LIN {X 0,Y 417.016,Z 398.719,A -85,B 0,C 180,E1 -10166.134,E2 -10166.134} C_VEL
LIN {X 0,Y 417.047,Z 400.246,A -85,B 0,C 180,E1 -10167.102,E2 -10167.102} C_VEL
LIN {X 0,Y 417.071,Z 401.315,A -85,B 0,C 180,E1 -10168.068,E2 -10168.068} C_VEL
LIN {X 0,Y 417.03,Z 402.263,A -85,B 0,C 180,E1 -10170,E2 -10170} C_VEL
LIN {X 0,Y 417.016,Z 402.15,A -85,B 0,C 180,E1 -10170.965,E2 -10170.965} C_VEL
LIN {X 0,Y 417.07,Z 401.605,A -85,B 0,C 180,E1 -10171.931,E2 -10171.931} C_VEL
LIN {X 0,Y 417.03,Z 400.658,A -85,B 0,C 180,E1 -10172.898,E2 -10172.898} C_VEL
LIN {X 0,Y 417.014,Z 399.317,A -85,B 0,C 180,E1 -10173.865,E2 -10173.865} C_VEL
LIN {X 0,Y 417.113,Z 396.49,A -85,B 0,C 180,E1 -10175.317,E2 -10175.317} C_VEL
LIN {X 0,Y 417.163,Z 392.636,A -85,B 0,C 180,E1 -10176.773,E2 -10176.773} C_VEL
LIN {X 0,Y 417.446,Z 387.665,A -85,B 0,C 180,E1 -10178.227,E2 -10178.227} C_VEL
LIN {X 0,Y 417.809,Z 381.424,A -85,B 0,C 180,E1 -10179.684,E2 -10179.684} C_VEL
LIN {X 0,Y 418.374,Z 373.662,A -85,B 0,C 180,E1 -10181.138,E2 -10181.138} C_VEL
LIN {X 0,Y 419.211,Z 363.972,A -85,B 0,C 180,E1 -10182.588,E2 -10182.588} C_VEL
LIN {X 0,Y 419.889,Z 353.988,A -85,B 0,C 180,E1 -10183.799,E2 -10183.799} C_VEL
LIN {X 0,Y 420.769,Z 342.734,A -85,B 0,C 180,E1 -10184.881,E2 -10184.881} C_VEL
LIN {X 0,Y 421.539,Z 331.733,A -85,B 0,C 180,E1 -10185.719,E2 -10185.719} C_VEL
LIN {X 0,Y 422.358,Z 319.563,A -85,B 0,C 180,E1 -10186.432,E2 -10186.432} C_VEL
LIN {X 0,Y 422.975,Z 306.851,A -85,B 0,C 180,E1 -10186.966,E2 -10186.966} C_VEL
LIN {X 0,Y 423.495,Z 293.508,A -85,B 0,C 180,E1 -10187.318,E2 -10187.318} C_VEL
LIN {X 0,Y 424.284,Z 215.513,A -85,B 0,C 180,E1 -10188.688,E2 -10188.688} C_VEL
LIN {X 0,Y 421.243,Z 196.282,A -85,B 0,C 180,E1 -10189.197,E2 -10189.197} C_VEL
LIN {X 0,Y 419.891,Z 188.95,A -85,B 0,C 180,E1 -10189.422,E2 -10189.422} C_VEL
LIN {X 0,Y 421.037,Z 171.63,A -85,B 0,C 180,E1 -10192.794,E2 -10192.794} C_VEL
LIN {X 0,Y 421.61,Z 163.663,A -85,B 0,C 180,E1 -10194.366,E2 -10194.366} C_VEL
LIN {X 0,Y 420.366,Z 155.936,A -85,B 0,C 180,E1 -10196.032,E2 -10196.032} C_VEL
LIN {X 0,Y 418.252,Z 146.389,A -85,B 0,C 180,E1 -10198.203,E2 -10198.203} C_VEL
LIN {X 0,Y 418.213,Z 146.395,A -85,B 0,C 180,E1 -10201.396,E2 -10201.396} C_VEL
LIN {X 0,Y 418.255,Z 146.379,A -85,B 0,C 180,E1 -10204.577,E2 -10204.577} C_VEL
LIN {X 0,Y 418.222,Z 146.388,A -85,B 0,C 180,E1 -10207.832,E2 -10207.832} C_VEL
LIN {X 0,Y 418.209,Z 146.385,A -85,B 0,C 180,E1 -10210.95,E2 -10210.95} C_VEL
LIN {X 0,Y 418.205,Z 146.389,A -85,B 0,C 180,E1 -10213.728,E2 -10213.728} C_VEL
LIN {X 0,Y 418.201,Z 146.391,A -85,B 0,C 180,E1 -10216.447,E2 -10216.447} C_VEL
LIN {X 0,Y 418.208,Z 146.39,A -85,B 0,C 180,E1 -10219.133,E2 -10219.133} C_VEL
LIN {X 0,Y 418.233,Z 146.387,A -85,B 0,C 180,E1 -10222.775,E2 -10222.775} C_VEL
LIN {X 0,Y 418.229,Z 146.384,A -85,B 0,C 180,E1 -10226.321,E2 -10226.321} C_VEL
LIN {X 0,Y 418.235,Z 146.38,A -85,B 0,C 180,E1 -10229.727,E2 -10229.727} C_VEL
LIN {X 0,Y 418.203,Z 146.384,A -85,B 0,C 180,E1 -10233.016,E2 -10233.016} C_VEL
LIN {X 0,Y 418.253,Z 146.386,A -85,B 0,C 180,E1 -10236.216,E2 -10236.216} C_VEL
LIN {X 0,Y 418.23,Z 146.385,A -85,B 0,C 180,E1 -10239.335,E2 -10239.335} C_VEL
LIN {X 0,Y 418.237,Z 146.383,A -85,B 0,C 180,E1 -10242.394,E2 -10242.394} C_VEL
LIN {X 0,Y 418.279,Z 146.38,A -85,B 0,C 180,E1 -10245.402,E2 -10245.402} C_VEL
LIN {X 0,Y 418.307,Z 146.379,A -85,B 0,C 180,E1 -10248.368,E2 -10248.368} C_VEL
LIN {X 0,Y 418.449,Z 146.356,A -85,B 0,C 180,E1 -10252.278,E2 -10252.278} C_VEL
LIN {X 0,Y 418.487,Z 146.355,A -85,B 0,C 180,E1 -10254.216,E2 -10254.216} C_VEL
LIN {X 0,Y 418.536,Z 146.349,A -85,B 0,C 180,E1 -10258.075,E2 -10258.075} C_VEL
LIN {X 0,Y 418.565,Z 146.342,A -85,B 0,C 180,E1 -10259.999,E2 -10259.999} C_VEL
LIN {X 0,Y 418.493,Z 146.351,A -85,B 0,C 180,E1 -10262.887,E2 -10262.887} C_VEL
LIN {X 0,Y 418.446,Z 146.353,A -85,B 0,C 180,E1 -10266.519,E2 -10266.519} C_VEL
LIN {X 0,Y 418.34,Z 146.369,A -85,B 0,C 180,E1 -10269.671,E2 -10269.671} C_VEL
LIN {X 0,Y 418.348,Z 146.376,A -85,B 0,C 180,E1 -10273,E2 -10273} C_VEL
LIN {X 0,Y 418.313,Z 146.378,A -85,B 0,C 180,E1 -10276.734,E2 -10276.734} C_VEL
LIN {X 0,Y 418.271,Z 146.382,A -85,B 0,C 180,E1 -10279.789,E2 -10279.789} C_VEL
LIN {X 0,Y 418.232,Z 146.387,A -85,B 0,C 180,E1 -10282.736,E2 -10282.736} C_VEL
LIN {X 0,Y 418.261,Z 146.383,A -85,B 0,C 180,E1 -10285.904,E2 -10285.904} C_VEL
LIN {X 0,Y 418.268,Z 146.385,A -85,B 0,C 180,E1 -10289.104,E2 -10289.104} C_VEL
LIN {X 0,Y 418.256,Z 146.386,A -85,B 0,C 180,E1 -10292.843,E2 -10292.843} C_VEL
LIN {X 0,Y 418.243,Z 146.391,A -85,B 0,C 180,E1 -10296.237,E2 -10296.237} C_VEL
LIN {X 0,Y 418.247,Z 146.387,A -85,B 0,C 180,E1 -10299.682,E2 -10299.682} C_VEL
LIN {X 0,Y 418.228,Z 146.392,A -85,B 0,C 180,E1 -10302.321,E2 -10302.321} C_VEL
LIN {X 0,Y 418.234,Z 146.39,A -85,B 0,C 180,E1 -10305.108,E2 -10305.108} C_VEL
LIN {X 0,Y 418.247,Z 146.493,A -85,B 0,C 180,E1 -10307.098,E2 -10307.098} C_VEL
LIN {X 0,Y 420.308,Z 156.513,A -85,B 0,C 180,E1 -10309.56,E2 -10309.56} C_VEL
LIN {X 0,Y 420.473,Z 161.32,A -85,B 0,C 180,E1 -10310.665,E2 -10310.665} C_VEL
LIN {X 0,Y 424.772,Z 180.68,A -85,B 0,C 180,E1 -10311.261,E2 -10311.261} C_VEL
LIN {X 0,Y 423.613,Z 268.691,A -85,B 0,C 180,E1 -10312.816,E2 -10312.816} C_VEL
LIN {X 0,Y 423.211,Z 281.385,A -85,B 0,C 180,E1 -10313.221,E2 -10313.221} C_VEL
LIN {X 0,Y 422.69,Z 294.104,A -85,B 0,C 180,E1 -10313.825,E2 -10313.825} C_VEL
LIN {X 0,Y 421.974,Z 306.065,A -85,B 0,C 180,E1 -10314.596,E2 -10314.596} C_VEL
LIN {X 0,Y 421.162,Z 317.748,A -85,B 0,C 180,E1 -10315.578,E2 -10315.578} C_VEL
LIN {X 0,Y 420.343,Z 328.498,A -85,B 0,C 180,E1 -10316.717,E2 -10316.717} C_VEL
LIN {X 0,Y 419.641,Z 337.311,A -85,B 0,C 180,E1 -10317.877,E2 -10317.877} C_VEL
LIN {X 0,Y 418.911,Z 345.664,A -85,B 0,C 180,E1 -10319.223,E2 -10319.223} C_VEL
LIN {X 0,Y 418.274,Z 353.696,A -85,B 0,C 180,E1 -10320.839,E2 -10320.839} C_VEL
LIN {X 0,Y 417.818,Z 359.91,A -85,B 0,C 180,E1 -10322.447,E2 -10322.447} C_VEL
LIN {X 0,Y 417.449,Z 364.645,A -85,B 0,C 180,E1 -10324.041,E2 -10324.041} C_VEL
LIN {X 0,Y 417.257,Z 367.76,A -85,B 0,C 180,E1 -10325.44,E2 -10325.44} C_VEL
LIN {X 0,Y 417.028,Z 370.384,A -85,B 0,C 180,E1 -10327.194,E2 -10327.194} C_VEL
LIN {X 0,Y 417.008,Z 371.33,A -85,B 0,C 180,E1 -10328.237,E2 -10328.237} C_VEL
LIN {X 0,Y 416.93,Z 371.775,A -85,B 0,C 180,E1 -10329.269,E2 -10329.269} C_VEL
LIN {X 0,Y 416.941,Z 371.672,A -85,B 0,C 180,E1 -10330.722,E2 -10330.722} C_VEL
LIN {X 0,Y 416.976,Z 370.485,A -85,B 0,C 180,E1 -10332.339,E2 -10332.339} C_VEL
LIN {X 0,Y 417.129,Z 368.427,A -85,B 0,C 180,E1 -10333.812,E2 -10333.812} C_VEL
LIN {X 0,Y 417.298,Z 365.169,A -85,B 0,C 180,E1 -10335.367,E2 -10335.367} C_VEL
LIN {X 0,Y 417.539,Z 360.89,A -85,B 0,C 180,E1 -10336.866,E2 -10336.866} C_VEL
LIN {X 0,Y 417.912,Z 354.367,A -85,B 0,C 180,E1 -10338.603,E2 -10338.603} C_VEL
LIN {X 0,Y 418.368,Z 347.237,A -85,B 0,C 180,E1 -10340.085,E2 -10340.085} C_VEL
LIN {X 0,Y 418.677,Z 342.718,A -85,B 0,C 180,E1 -10340.871,E2 -10340.871} C_VEL
LIN {X 0,Y 418.226,Z 338.947,A -85,B 0,C 180,E1 -10341.486,E2 -10341.486} C_VEL
LIN {X 0,Y 415.824,Z 332.509,A -85,B 0,C 180,E1 -10342.469,E2 -10342.469} C_VEL
LIN {X 0,Y 413.531,Z 325.54,A -85,B 0,C 180,E1 -10343.39,E2 -10343.39} C_VEL
LIN {X 0,Y 413.248,Z 320.905,A -85,B 0,C 180,E1 -10343.904,E2 -10343.904} C_VEL
LIN {X 0,Y 413.946,Z 310.162,A -85,B 0,C 180,E1 -10344.886,E2 -10344.886} C_VEL
LIN {X 0,Y 414.53,Z 298.105,A -85,B 0,C 180,E1 -10345.746,E2 -10345.746} C_VEL
LIN {X 0,Y 415.093,Z 284.913,A -85,B 0,C 180,E1 -10346.448,E2 -10346.448} C_VEL
LIN {X 0,Y 415.474,Z 272.537,A -85,B 0,C 180,E1 -10346.899,E2 -10346.899} C_VEL
LIN {X 0,Y 415.743,Z 256.003,A -85,B 0,C 180,E1 -10347.248,E2 -10347.248} C_VEL
LIN {X 0,Y 416.545,Z 180.606,A -85,B 0,C 180,E1 -10348.565,E2 -10348.565} C_VEL
LIN {X 0,Y 412.854,Z 161.197,A -85,B 0,C 180,E1 -10349.086,E2 -10349.086} C_VEL
LIN {X 0,Y 412.939,Z 156.063,A -85,B 0,C 180,E1 -10350.244,E2 -10350.244} C_VEL
LIN {X 0,Y 411.456,Z 147.236,A -85,B 0,C 180,E1 -10352.386,E2 -10352.386} C_VEL
LIN {X 0,Y 411.411,Z 147.241,A -85,B 0,C 180,E1 -10355.883,E2 -10355.883} C_VEL
LIN {X 0,Y 411.302,Z 147.247,A -85,B 0,C 180,E1 -10358.847,E2 -10358.847} C_VEL
LIN {X 0,Y 411.266,Z 147.259,A -85,B 0,C 180,E1 -10361.834,E2 -10361.834} C_VEL
LIN {X 0,Y 411.203,Z 147.26,A -85,B 0,C 180,E1 -10364.855,E2 -10364.855} C_VEL
LIN {X 0,Y 411.17,Z 147.268,A -85,B 0,C 180,E1 -10367.919,E2 -10367.919} C_VEL
LIN {X 0,Y 411.175,Z 147.265,A -85,B 0,C 180,E1 -10371.036,E2 -10371.036} C_VEL
LIN {X 0,Y 411.167,Z 147.265,A -85,B 0,C 180,E1 -10374.219,E2 -10374.219} C_VEL
LIN {X 0,Y 411.137,Z 147.274,A -85,B 0,C 180,E1 -10377.487,E2 -10377.487} C_VEL
LIN {X 0,Y 411.189,Z 147.264,A -85,B 0,C 180,E1 -10379.714,E2 -10379.714} C_VEL
LIN {X 0,Y 411.2,Z 147.266,A -85,B 0,C 180,E1 -10383.157,E2 -10383.157} C_VEL
LIN {X 0,Y 411.185,Z 147.263,A -85,B 0,C 180,E1 -10386.552,E2 -10386.552} C_VEL
LIN {X 0,Y 411.165,Z 147.266,A -85,B 0,C 180,E1 -10389.721,E2 -10389.721} C_VEL
LIN {X 0,Y 411.159,Z 147.271,A -85,B 0,C 180,E1 -10393.136,E2 -10393.136} C_VEL
LIN {X 0,Y 411.162,Z 147.265,A -85,B 0,C 180,E1 -10395.883,E2 -10395.883} C_VEL
LIN {X 0,Y 411.157,Z 147.266,A -85,B 0,C 180,E1 -10399.494,E2 -10399.494} C_VEL
LIN {X 0,Y 411.181,Z 147.263,A -85,B 0,C 180,E1 -10402.026,E2 -10402.026} C_VEL
LIN {X 0,Y 411.2,Z 147.263,A -85,B 0,C 180,E1 -10405.125,E2 -10405.125} C_VEL
LIN {X 0,Y 411.154,Z 147.267,A -85,B 0,C 180,E1 -10408.002,E2 -10408.002} C_VEL
LIN {X 0,Y 411.168,Z 147.264,A -85,B 0,C 180,E1 -10411.407,E2 -10411.407} C_VEL
LIN {X 0,Y 411.188,Z 147.264,A -85,B 0,C 180,E1 -10414.942,E2 -10414.942} C_VEL
LIN {X 0,Y 411.198,Z 147.263,A -85,B 0,C 180,E1 -10417.914,E2 -10417.914} C_VEL
LIN {X 0,Y 411.18,Z 147.263,A -85,B 0,C 180,E1 -10421.05,E2 -10421.05} C_VEL
LIN {X 0,Y 411.199,Z 147.266,A -85,B 0,C 180,E1 -10424.13,E2 -10424.13} C_VEL
LIN {X 0,Y 411.299,Z 147.248,A -85,B 0,C 180,E1 -10427.166,E2 -10427.166} C_VEL
LIN {X 0,Y 411.278,Z 147.257,A -85,B 0,C 180,E1 -10430.161,E2 -10430.161} C_VEL
LIN {X 0,Y 411.394,Z 147.236,A -85,B 0,C 180,E1 -10433.132,E2 -10433.132} C_VEL
LIN {X 0,Y 411.288,Z 147.249,A -85,B 0,C 180,E1 -10435.099,E2 -10435.099} C_VEL
LIN {X 0,Y 411.506,Z 147.227,A -85,B 0,C 180,E1 -10438.043,E2 -10438.043} C_VEL
LIN {X 0,Y 411.381,Z 147.238,A -85,B 0,C 180,E1 -10440.979,E2 -10440.979} C_VEL
LIN {X 0,Y 411.43,Z 147.232,A -85,B 0,C 180,E1 -10442.938,E2 -10442.938} C_VEL
LIN {X 0,Y 411.393,Z 147.236,A -85,B 0,C 180,E1 -10446.869,E2 -10446.869} C_VEL
LIN {X 0,Y 411.287,Z 147.254,A -85,B 0,C 180,E1 -10449.839,E2 -10449.839} C_VEL
LIN {X 0,Y 411.311,Z 147.249,A -85,B 0,C 180,E1 -10453.104,E2 -10453.104} C_VEL
LIN {X 0,Y 411.215,Z 147.26,A -85,B 0,C 180,E1 -10456.891,E2 -10456.891} C_VEL
LIN {X 0,Y 411.215,Z 147.259,A -85,B 0,C 180,E1 -10459.988,E2 -10459.988} C_VEL
LIN {X 0,Y 411.192,Z 147.267,A -85,B 0,C 180,E1 -10463.149,E2 -10463.149} C_VEL
LIN {X 0,Y 411.176,Z 147.263,A -85,B 0,C 180,E1 -10466.386,E2 -10466.386} C_VEL
LIN {X 0,Y 411.199,Z 147.261,A -85,B 0,C 180,E1 -10469.713,E2 -10469.713} C_VEL
LIN {X 0,Y 411.209,Z 147.264,A -85,B 0,C 180,E1 -10473.156,E2 -10473.156} C_VEL
LIN {X 0,Y 411.196,Z 147.264,A -85,B 0,C 180,E1 -10476.552,E2 -10476.552} C_VEL
LIN {X 0,Y 411.182,Z 147.263,A -85,B 0,C 180,E1 -10479.722,E2 -10479.722} C_VEL
LIN {X 0,Y 411.166,Z 147.267,A -85,B 0,C 180,E1 -10483.135,E2 -10483.135} C_VEL
LIN {X 0,Y 411.168,Z 147.264,A -85,B 0,C 180,E1 -10485.882,E2 -10485.882} C_VEL
LIN {X 0,Y 411.162,Z 147.265,A -85,B 0,C 180,E1 -10489.493,E2 -10489.493} C_VEL
LIN {X 0,Y 411.19,Z 147.263,A -85,B 0,C 180,E1 -10492.025,E2 -10492.025} C_VEL
LIN {X 0,Y 411.207,Z 147.26,A -85,B 0,C 180,E1 -10495.123,E2 -10495.123} C_VEL
LIN {X 0,Y 411.168,Z 147.267,A -85,B 0,C 180,E1 -10498.002,E2 -10498.002} C_VEL
LIN {X 0,Y 411.2,Z 147.264,A -85,B 0,C 180,E1 -10501.408,E2 -10501.408} C_VEL
LIN {X 0,Y 411.229,Z 147.314,A -85,B 0,C 180,E1 -10502.451,E2 -10502.451} C_VEL
LIN {X 0,Y 413.944,Z 161.206,A -85,B 0,C 180,E1 -10505.42,E2 -10505.42} C_VEL
LIN {X 0,Y 413.846,Z 166.622,A -85,B 0,C 180,E1 -10506.498,E2 -10506.498} C_VEL
LIN {X 0,Y 412.705,Z 184.992,A -85,B 0,C 180,E1 -10510.087,E2 -10510.087} C_VEL
LIN {X 0,Y 412.413,Z 189.335,A -85,B 0,C 180,E1 -10510.929,E2 -10510.929} C_VEL
LIN {X 0,Y 416.326,Z 217.289,A -85,B 0,C 180,E1 -10511.589,E2 -10511.589} C_VEL
LIN {X 0,Y 415.353,Z 298.398,A -85,B 0,C 180,E1 -10513.029,E2 -10513.029} C_VEL
LIN {X 0,Y 414.814,Z 312.207,A -85,B 0,C 180,E1 -10513.482,E2 -10513.482} C_VEL
LIN {X 0,Y 414.202,Z 325.137,A -85,B 0,C 180,E1 -10514.121,E2 -10514.121} C_VEL
LIN {X 0,Y 413.45,Z 337.732,A -85,B 0,C 180,E1 -10514.976,E2 -10514.976} C_VEL
LIN {X 0,Y 412.691,Z 349.444,A -85,B 0,C 180,E1 -10516.003,E2 -10516.003} C_VEL
LIN {X 0,Y 411.952,Z 360.048,A -85,B 0,C 180,E1 -10517.186,E2 -10517.186} C_VEL
LIN {X 0,Y 411.37,Z 369.023,A -85,B 0,C 180,E1 -10518.419,E2 -10518.419} C_VEL
LIN {X 0,Y 410.782,Z 377.769,A -85,B 0,C 180,E1 -10519.9,E2 -10519.9} C_VEL
LIN {X 0,Y 410.39,Z 384.734,A -85,B 0,C 180,E1 -10521.382,E2 -10521.382} C_VEL
LIN {X 0,Y 410.095,Z 391.121,A -85,B 0,C 180,E1 -10523.11,E2 -10523.11} C_VEL
LIN {X 0,Y 410.004,Z 395.299,A -85,B 0,C 180,E1 -10524.59,E2 -10524.59} C_VEL
LIN {X 0,Y 409.935,Z 398.402,A -85,B 0,C 180,E1 -10526.068,E2 -10526.068} C_VEL
LIN {X 0,Y 409.946,Z 399.944,A -85,B 0,C 180,E1 -10527.052,E2 -10527.052} C_VEL
LIN {X 0,Y 409.999,Z 401.03,A -85,B 0,C 180,E1 -10528.035,E2 -10528.035} C_VEL
LIN {X 0,Y 409.951,Z 401.998,A -85,B 0,C 180,E1 -10530,E2 -10530} C_VEL
LIN {X 0,Y 409.941,Z 401.899,A -85,B 0,C 180,E1 -10530.982,E2 -10530.982} C_VEL
LIN {X 0,Y 409.997,Z 401.37,A -85,B 0,C 180,E1 -10531.965,E2 -10531.965} C_VEL
LIN {X 0,Y 409.932,Z 399.1,A -85,B 0,C 180,E1 -10533.932,E2 -10533.932} C_VEL
LIN {X 0,Y 410.006,Z 396.296,A -85,B 0,C 180,E1 -10535.41,E2 -10535.41} C_VEL
LIN {X 0,Y 410.084,Z 392.472,A -85,B 0,C 180,E1 -10536.89,E2 -10536.89} C_VEL
LIN {X 0,Y 410.402,Z 387.537,A -85,B 0,C 180,E1 -10538.37,E2 -10538.37} C_VEL
LIN {X 0,Y 410.786,Z 381.34,A -85,B 0,C 180,E1 -10539.851,E2 -10539.851} C_VEL
LIN {X 0,Y 411.396,Z 373.648,A -85,B 0,C 180,E1 -10541.33,E2 -10541.33} C_VEL
LIN {X 0,Y 412.279,Z 364.011,A -85,B 0,C 180,E1 -10542.803,E2 -10542.803} C_VEL
LIN {X 0,Y 413.037,Z 353.536,A -85,B 0,C 180,E1 -10544.097,E2 -10544.097} C_VEL
LIN {X 0,Y 413.907,Z 342.952,A -85,B 0,C 180,E1 -10545.133,E2 -10545.133} C_VEL
LIN {X 0,Y 414.73,Z 332.065,A -85,B 0,C 180,E1 -10545.984,E2 -10545.984} C_VEL
LIN {X 0,Y 415.571,Z 320.062,A -85,B 0,C 180,E1 -10546.708,E2 -10546.708} C_VEL
LIN {X 0,Y 416.233,Z 307.801,A -85,B 0,C 180,E1 -10547.25,E2 -10547.25} C_VEL
LIN {X 0,Y 416.793,Z 295.256,A -85,B 0,C 180,E1 -10547.606,E2 -10547.606} C_VEL
LIN {X 0,Y 417.68,Z 216.545,A -85,B 0,C 180,E1 -10549.016,E2 -10549.016} C_VEL
LIN {X 0,Y 414.773,Z 197.99,A -85,B 0,C 180,E1 -10549.517,E2 -10549.517} C_VEL
LIN {X 0,Y 413.015,Z 188.743,A -85,B 0,C 180,E1 -10549.791,E2 -10549.791} C_VEL
LIN {X 0,Y 414.291,Z 170.892,A -85,B 0,C 180,E1 -10553.338,E2 -10553.338} C_VEL
LIN {X 0,Y 414.728,Z 164.974,A -85,B 0,C 180,E1 -10554.531,E2 -10554.531} C_VEL
LIN {X 0,Y 413.149,Z 155.963,A -85,B 0,C 180,E1 -10556.522,E2 -10556.522} C_VEL
LIN {X 0,Y 411.244,Z 147.262,A -85,B 0,C 180,E1 -10558.553,E2 -10558.553} C_VEL
LIN {X 0,Y 411.167,Z 147.268,A -85,B 0,C 180,E1 -10561.997,E2 -10561.997} C_VEL
LIN {X 0,Y 411.205,Z 147.259,A -85,B 0,C 180,E1 -10564.876,E2 -10564.876} C_VEL
LIN {X 0,Y 411.195,Z 147.264,A -85,B 0,C 180,E1 -10568.166,E2 -10568.166} C_VEL
LIN {X 0,Y 411.162,Z 147.268,A -85,B 0,C 180,E1 -10571.807,E2 -10571.807} C_VEL
LIN {X 0,Y 411.176,Z 147.267,A -85,B 0,C 180,E1 -10575.509,E2 -10575.509} C_VEL
LIN {X 0,Y 411.148,Z 147.271,A -85,B 0,C 180,E1 -10578.774,E2 -10578.774} C_VEL
LIN {X 0,Y 411.181,Z 147.262,A -85,B 0,C 180,E1 -10582.024,E2 -10582.024} C_VEL
LIN {X 0,Y 411.201,Z 147.259,A -85,B 0,C 180,E1 -10585.124,E2 -10585.124} C_VEL
LIN {X 0,Y 411.155,Z 147.267,A -85,B 0,C 180,E1 -10588.001,E2 -10588.001} C_VEL
LIN {X 0,Y 411.169,Z 147.264,A -85,B 0,C 180,E1 -10591.406,E2 -10591.406} C_VEL
LIN {X 0,Y 411.189,Z 147.264,A -85,B 0,C 180,E1 -10594.941,E2 -10594.941} C_VEL
LIN {X 0,Y 411.198,Z 147.255,A -85,B 0,C 180,E1 -10597.913,E2 -10597.913} C_VEL
LIN {X 0,Y 411.18,Z 147.261,A -85,B 0,C 180,E1 -10601.049,E2 -10601.049} C_VEL
LIN {X 0,Y 411.211,Z 147.264,A -85,B 0,C 180,E1 -10604.129,E2 -10604.129} C_VEL
LIN {X 0,Y 411.305,Z 147.24,A -85,B 0,C 180,E1 -10607.165,E2 -10607.165} C_VEL
LIN {X 0,Y 411.282,Z 147.252,A -85,B 0,C 180,E1 -10610.16,E2 -10610.16} C_VEL
LIN {X 0,Y 411.393,Z 147.234,A -85,B 0,C 180,E1 -10613.131,E2 -10613.131} C_VEL
LIN {X 0,Y 411.293,Z 147.249,A -85,B 0,C 180,E1 -10615.098,E2 -10615.098} C_VEL
LIN {X 0,Y 411.505,Z 147.225,A -85,B 0,C 180,E1 -10618.042,E2 -10618.042} C_VEL
LIN {X 0,Y 411.517,Z 147.22,A -85,B 0,C 180,E1 -10619.999,E2 -10619.999} C_VEL
LIN {X 0,Y 411.45,Z 147.228,A -85,B 0,C 180,E1 -10622.937,E2 -10622.937} C_VEL
LIN {X 0,Y 411.396,Z 147.231,A -85,B 0,C 180,E1 -10626.516,E2 -10626.516} C_VEL
LIN {X 0,Y 411.321,Z 147.248,A -85,B 0,C 180,E1 -10628.845,E2 -10628.845} C_VEL
LIN {X 0,Y 411.285,Z 147.252,A -85,B 0,C 180,E1 -10631.832,E2 -10631.832} C_VEL
LIN {X 0,Y 411.26,Z 147.252,A -85,B 0,C 180,E1 -10634.852,E2 -10634.852} C_VEL
LIN {X 0,Y 411.246,Z 147.252,A -85,B 0,C 180,E1 -10637.915,E2 -10637.915} C_VEL
LIN {X 0,Y 411.197,Z 147.264,A -85,B 0,C 180,E1 -10641.033,E2 -10641.033} C_VEL
LIN {X 0,Y 411.212,Z 147.263,A -85,B 0,C 180,E1 -10644.216,E2 -10644.216} C_VEL
LIN {X 0,Y 411.258,Z 147.254,A -85,B 0,C 180,E1 -10647.477,E2 -10647.477} C_VEL
LIN {X 0,Y 411.189,Z 147.266,A -85,B 0,C 180,E1 -10650.847,E2 -10650.847} C_VEL
LIN {X 0,Y 411.204,Z 147.266,A -85,B 0,C 180,E1 -10654.333,E2 -10654.333} C_VEL
LIN {X 0,Y 411.193,Z 147.269,A -85,B 0,C 180,E1 -10657.973,E2 -10657.973} C_VEL
LIN {X 0,Y 411.162,Z 147.272,A -85,B 0,C 180,E1 -10661.228,E2 -10661.228} C_VEL
LIN {X 0,Y 411.174,Z 147.269,A -85,B 0,C 180,E1 -10664.49,E2 -10664.49} C_VEL
LIN {X 0,Y 411.201,Z 147.42,A -85,B 0,C 180,E1 -10666.786,E2 -10666.786} C_VEL
LIN {X 0,Y 413.234,Z 156.771,A -85,B 0,C 180,E1 -10669.136,E2 -10669.136} C_VEL
LIN {X 0,Y 413.636,Z 161.696,A -85,B 0,C 180,E1 -10670.296,E2 -10670.296} C_VEL
LIN {X 0,Y 418.162,Z 181.697,A -85,B 0,C 180,E1 -10670.923,E2 -10670.923} C_VEL
LIN {X 0,Y 416.952,Z 268.815,A -85,B 0,C 180,E1 -10672.485,E2 -10672.485} C_VEL
LIN {X 0,Y 416.527,Z 281.651,A -85,B 0,C 180,E1 -10672.9,E2 -10672.9} C_VEL
LIN {X 0,Y 415.972,Z 294.535,A -85,B 0,C 180,E1 -10673.522,E2 -10673.522} C_VEL
LIN {X 0,Y 415.244,Z 306.088,A -85,B 0,C 180,E1 -10674.277,E2 -10674.277} C_VEL
LIN {X 0,Y 414.401,Z 317.375,A -85,B 0,C 180,E1 -10675.232,E2 -10675.232} C_VEL
LIN {X 0,Y 413.546,Z 328.154,A -85,B 0,C 180,E1 -10676.379,E2 -10676.379} C_VEL
LIN {X 0,Y 412.802,Z 337.174,A -85,B 0,C 180,E1 -10677.568,E2 -10677.568} C_VEL
LIN {X 0,Y 411.99,Z 345.853,A -85,B 0,C 180,E1 -10678.983,E2 -10678.983} C_VEL
LIN {X 0,Y 411.302,Z 353.904,A -85,B 0,C 180,E1 -10680.626,E2 -10680.626} C_VEL
LIN {X 0,Y 410.867,Z 359.031,A -85,B 0,C 180,E1 -10681.94,E2 -10681.94} C_VEL
LIN {X 0,Y 410.476,Z 364.076,A -85,B 0,C 180,E1 -10683.566,E2 -10683.566} C_VEL
LIN {X 0,Y 410.193,Z 367.874,A -85,B 0,C 180,E1 -10685.238,E2 -10685.238} C_VEL
LIN {X 0,Y 409.975,Z 370.277,A -85,B 0,C 180,E1 -10686.779,E2 -10686.779} C_VEL
LIN {X 0,Y 409.922,Z 371.331,A -85,B 0,C 180,E1 -10687.841,E2 -10687.841} C_VEL
LIN {X 0,Y 409.851,Z 371.951,A -85,B 0,C 180,E1 -10688.894,E2 -10688.894} C_VEL
LIN {X 0,Y 409.841,Z 371.981,A -85,B 0,C 180,E1 -10690.585,E2 -10690.585} C_VEL
LIN {X 0,Y 409.855,Z 371.066,A -85,B 0,C 180,E1 -10692.022,E2 -10692.022} C_VEL
LIN {X 0,Y 410.021,Z 368.916,A -85,B 0,C 180,E1 -10693.711,E2 -10693.711} C_VEL
LIN {X 0,Y 410.175,Z 366.174,A -85,B 0,C 180,E1 -10695.107,E2 -10695.107} C_VEL
LIN {X 0,Y 410.431,Z 362.134,A -85,B 0,C 180,E1 -10696.634,E2 -10696.634} C_VEL
LIN {X 0,Y 410.769,Z 355.898,A -85,B 0,C 180,E1 -10698.403,E2 -10698.403} C_VEL
LIN {X 0,Y 411.242,Z 349.058,A -85,B 0,C 180,E1 -10699.912,E2 -10699.912} C_VEL
LIN {X 0,Y 411.779,Z 340.961,A -85,B 0,C 180,E1 -10701.35,E2 -10701.35} C_VEL
LIN {X 0,Y 412.453,Z 331.79,A -85,B 0,C 180,E1 -10702.658,E2 -10702.658} C_VEL
LIN {X 0,Y 413.248,Z 320.905,A -85,B 0,C 180,E1 -10703.904,E2 -10703.904} C_VEL
LIN {X 0,Y 412.997,Z 316.162,A -85,B 0,C 180,E1 -10704.39,E2 -10704.39} C_VEL
LIN {X 0,Y 410.816,Z 308.258,A -85,B 0,C 180,E1 -10705.162,E2 -10705.162} C_VEL
LIN {X 0,Y 408.417,Z 299.974,A -85,B 0,C 180,E1 -10705.851,E2 -10705.851} C_VEL
LIN {X 0,Y 407.822,Z 294.631,A -85,B 0,C 180,E1 -10706.2,E2 -10706.2} C_VEL
LIN {X 0,Y 408.289,Z 281.842,A -85,B 0,C 180,E1 -10706.827,E2 -10706.827} C_VEL
LIN {X 0,Y 408.714,Z 268.82,A -85,B 0,C 180,E1 -10707.253,E2 -10707.253} C_VEL
LIN {X 0,Y 409.74,Z 181.606,A -85,B 0,C 180,E1 -10708.824,E2 -10708.824} C_VEL
LIN {X 0,Y 405.895,Z 161.458,A -85,B 0,C 180,E1 -10709.368,E2 -10709.368} C_VEL
LIN {X 0,Y 405.861,Z 156.573,A -85,B 0,C 180,E1 -10710.496,E2 -10710.496} C_VEL
LIN {X 0,Y 404.424,Z 148.113,A -85,B 0,C 180,E1 -10712.584,E2 -10712.584} C_VEL
LIN {X 0,Y 404.361,Z 148.119,A -85,B 0,C 180,E1 -10715.986,E2 -10715.986} C_VEL
LIN {X 0,Y 404.251,Z 148.126,A -85,B 0,C 180,E1 -10719.002,E2 -10719.002} C_VEL
LIN {X 0,Y 404.241,Z 148.131,A -85,B 0,C 180,E1 -10722.042,E2 -10722.042} C_VEL
LIN {X 0,Y 404.152,Z 148.139,A -85,B 0,C 180,E1 -10725.12,E2 -10725.12} C_VEL
LIN {X 0,Y 404.128,Z 148.142,A -85,B 0,C 180,E1 -10728.242,E2 -10728.242} C_VEL
LIN {X 0,Y 404.121,Z 148.148,A -85,B 0,C 180,E1 -10731.421,E2 -10731.421} C_VEL
LIN {X 0,Y 404.123,Z 148.142,A -85,B 0,C 180,E1 -10734.67,E2 -10734.67} C_VEL
LIN {X 0,Y 404.095,Z 148.146,A -85,B 0,C 180,E1 -10738.008,E2 -10738.008} C_VEL
LIN {X 0,Y 404.135,Z 148.14,A -85,B 0,C 180,E1 -10740.286,E2 -10740.286} C_VEL
LIN {X 0,Y 404.133,Z 148.142,A -85,B 0,C 180,E1 -10743.814,E2 -10743.814} C_VEL
LIN {X 0,Y 404.128,Z 148.145,A -85,B 0,C 180,E1 -10746.874,E2 -10746.874} C_VEL
LIN {X 0,Y 404.115,Z 148.143,A -85,B 0,C 180,E1 -10750.076,E2 -10750.076} C_VEL
LIN {X 0,Y 404.139,Z 148.146,A -85,B 0,C 180,E1 -10753.082,E2 -10753.082} C_VEL
LIN {X 0,Y 404.119,Z 148.142,A -85,B 0,C 180,E1 -10755.923,E2 -10755.923} C_VEL
LIN {X 0,Y 404.101,Z 148.149,A -85,B 0,C 180,E1 -10758.633,E2 -10758.633} C_VEL
LIN {X 0,Y 404.137,Z 148.141,A -85,B 0,C 180,E1 -10761.496,E2 -10761.496} C_VEL
LIN {X 0,Y 404.171,Z 148.14,A -85,B 0,C 180,E1 -10764.983,E2 -10764.983} C_VEL
LIN {X 0,Y 404.131,Z 148.146,A -85,B 0,C 180,E1 -10768.445,E2 -10768.445} C_VEL
LIN {X 0,Y 404.147,Z 148.142,A -85,B 0,C 180,E1 -10770.863,E2 -10770.863} C_VEL
LIN {X 0,Y 404.152,Z 148.142,A -85,B 0,C 180,E1 -10774.724,E2 -10774.724} C_VEL
LIN {X 0,Y 404.164,Z 148.137,A -85,B 0,C 180,E1 -10777.508,E2 -10777.508} C_VEL
LIN {X 0,Y 404.133,Z 148.143,A -85,B 0,C 180,E1 -10780.707,E2 -10780.707} C_VEL
LIN {X 0,Y 404.173,Z 148.138,A -85,B 0,C 180,E1 -10783.847,E2 -10783.847} C_VEL
LIN {X 0,Y 404.267,Z 148.124,A -85,B 0,C 180,E1 -10786.939,E2 -10786.939} C_VEL
LIN {X 0,Y 404.246,Z 148.132,A -85,B 0,C 180,E1 -10789.989,E2 -10789.989} C_VEL
LIN {X 0,Y 404.344,Z 148.114,A -85,B 0,C 180,E1 -10793.012,E2 -10793.012} C_VEL
LIN {X 0,Y 404.259,Z 148.125,A -85,B 0,C 180,E1 -10795.014,E2 -10795.014} C_VEL
LIN {X 0,Y 404.474,Z 148.104,A -85,B 0,C 180,E1 -10798.009,E2 -10798.009} C_VEL
LIN {X 0,Y 404.351,Z 148.114,A -85,B 0,C 180,E1 -10800.996,E2 -10800.996} C_VEL
LIN {X 0,Y 404.39,Z 148.109,A -85,B 0,C 180,E1 -10802.989,E2 -10802.989} C_VEL
LIN {X 0,Y 404.343,Z 148.115,A -85,B 0,C 180,E1 -10806.989,E2 -10806.989} C_VEL
LIN {X 0,Y 404.254,Z 148.128,A -85,B 0,C 180,E1 -10810.012,E2 -10810.012} C_VEL
LIN {X 0,Y 404.272,Z 148.127,A -85,B 0,C 180,E1 -10813.212,E2 -10813.212} C_VEL
LIN {X 0,Y 404.183,Z 148.139,A -85,B 0,C 180,E1 -10817.194,E2 -10817.194} C_VEL
LIN {X 0,Y 404.16,Z 148.137,A -85,B 0,C 180,E1 -10820.352,E2 -10820.352} C_VEL
LIN {X 0,Y 404.153,Z 148.141,A -85,B 0,C 180,E1 -10823.576,E2 -10823.576} C_VEL
LIN {X 0,Y 404.108,Z 148.147,A -85,B 0,C 180,E1 -10826.884,E2 -10826.884} C_VEL
LIN {X 0,Y 404.146,Z 148.139,A -85,B 0,C 180,E1 -10830.286,E2 -10830.286} C_VEL
LIN {X 0,Y 404.142,Z 148.14,A -85,B 0,C 180,E1 -10833.813,E2 -10833.813} C_VEL
LIN {X 0,Y 404.14,Z 148.146,A -85,B 0,C 180,E1 -10836.875,E2 -10836.875} C_VEL
LIN {X 0,Y 404.121,Z 148.142,A -85,B 0,C 180,E1 -10840.075,E2 -10840.075} C_VEL
LIN {X 0,Y 404.146,Z 148.142,A -85,B 0,C 180,E1 -10843.082,E2 -10843.082} C_VEL
LIN {X 0,Y 404.125,Z 148.142,A -85,B 0,C 180,E1 -10845.922,E2 -10845.922} C_VEL
LIN {X 0,Y 404.106,Z 148.151,A -85,B 0,C 180,E1 -10848.633,E2 -10848.633} C_VEL
LIN {X 0,Y 404.144,Z 148.139,A -85,B 0,C 180,E1 -10851.495,E2 -10851.495} C_VEL
LIN {X 0,Y 404.182,Z 148.136,A -85,B 0,C 180,E1 -10854.983,E2 -10854.983} C_VEL
LIN {X 0,Y 404.143,Z 148.146,A -85,B 0,C 180,E1 -10858.442,E2 -10858.442} C_VEL
LIN {X 0,Y 404.199,Z 148.142,A -85,B 0,C 180,E1 -10862,E2 -10862} C_VEL
LIN {X 0,Y 404.192,Z 148.259,A -85,B 0,C 180,E1 -10862.246,E2 -10862.246} C_VEL
LIN {X 0,Y 406.885,Z 162.001,A -85,B 0,C 180,E1 -10865.237,E2 -10865.237} C_VEL
LIN {X 0,Y 407.035,Z 165.534,A -85,B 0,C 180,E1 -10865.964,E2 -10865.964} C_VEL
LIN {X 0,Y 405.998,Z 179.218,A -85,B 0,C 180,E1 -10868.683,E2 -10868.683} C_VEL
LIN {X 0,Y 405.464,Z 189.048,A -85,B 0,C 180,E1 -10870.627,E2 -10870.627} C_VEL
LIN {X 0,Y 409.488,Z 217.559,A -85,B 0,C 180,E1 -10871.326,E2 -10871.326} C_VEL
LIN {X 0,Y 408.506,Z 297.62,A -85,B 0,C 180,E1 -10872.768,E2 -10872.768} C_VEL
LIN {X 0,Y 407.996,Z 310.838,A -85,B 0,C 180,E1 -10873.198,E2 -10873.198} C_VEL
LIN {X 0,Y 407.393,Z 323.009,A -85,B 0,C 180,E1 -10873.784,E2 -10873.784} C_VEL
LIN {X 0,Y 406.625,Z 335.295,A -85,B 0,C 180,E1 -10874.589,E2 -10874.589} C_VEL
LIN {X 0,Y 405.857,Z 346.933,A -85,B 0,C 180,E1 -10875.586,E2 -10875.586} C_VEL
LIN {X 0,Y 405.152,Z 357.815,A -85,B 0,C 180,E1 -10876.76,E2 -10876.76} C_VEL
LIN {X 0,Y 404.536,Z 366.825,A -85,B 0,C 180,E1 -10877.967,E2 -10877.967} C_VEL
LIN {X 0,Y 403.81,Z 375.914,A -85,B 0,C 180,E1 -10879.47,E2 -10879.47} C_VEL
LIN {X 0,Y 403.378,Z 383.237,A -85,B 0,C 180,E1 -10880.978,E2 -10880.978} C_VEL
LIN {X 0,Y 403.11,Z 389.088,A -85,B 0,C 180,E1 -10882.486,E2 -10882.486} C_VEL
LIN {X 0,Y 402.94,Z 393.68,A -85,B 0,C 180,E1 -10883.993,E2 -10883.993} C_VEL
LIN {X 0,Y 402.938,Z 396.098,A -85,B 0,C 180,E1 -10884.997,E2 -10884.997} C_VEL
LIN {X 0,Y 402.856,Z 398.071,A -85,B 0,C 180,E1 -10885.998,E2 -10885.998} C_VEL
LIN {X 0,Y 402.846,Z 399.629,A -85,B 0,C 180,E1 -10887,E2 -10887} C_VEL
LIN {X 0,Y 402.91,Z 400.739,A -85,B 0,C 180,E1 -10888.001,E2 -10888.001} C_VEL
LIN {X 0,Y 402.884,Z 401.43,A -85,B 0,C 180,E1 -10889,E2 -10889} C_VEL
LIN {X 0,Y 402.875,Z 401.732,A -85,B 0,C 180,E1 -10890,E2 -10890} C_VEL
LIN {X 0,Y 402.868,Z 401.646,A -85,B 0,C 180,E1 -10890.999,E2 -10890.999} C_VEL
LIN {X 0,Y 402.907,Z 401.141,A -85,B 0,C 180,E1 -10891.999,E2 -10891.999} C_VEL
LIN {X 0,Y 402.852,Z 398.901,A -85,B 0,C 180,E1 -10894.001,E2 -10894.001} C_VEL
LIN {X 0,Y 402.899,Z 396.125,A -85,B 0,C 180,E1 -10895.505,E2 -10895.505} C_VEL
LIN {X 0,Y 403.033,Z 392.333,A -85,B 0,C 180,E1 -10897.011,E2 -10897.011} C_VEL
LIN {X 0,Y 403.346,Z 387.429,A -85,B 0,C 180,E1 -10898.517,E2 -10898.517} C_VEL
LIN {X 0,Y 403.779,Z 381.267,A -85,B 0,C 180,E1 -10900.024,E2 -10900.024} C_VEL
LIN {X 0,Y 404.399,Z 373.627,A -85,B 0,C 180,E1 -10901.529,E2 -10901.529} C_VEL
LIN {X 0,Y 405.174,Z 365.829,A -85,B 0,C 180,E1 -10902.777,E2 -10902.777} C_VEL
LIN {X 0,Y 405.887,Z 356.331,A -85,B 0,C 180,E1 -10904.029,E2 -10904.029} C_VEL
LIN {X 0,Y 406.833,Z 345.821,A -85,B 0,C 180,E1 -10905.146,E2 -10905.146} C_VEL
LIN {X 0,Y 407.814,Z 334.14,A -85,B 0,C 180,E1 -10906.134,E2 -10906.134} C_VEL
LIN {X 0,Y 408.691,Z 322.804,A -85,B 0,C 180,E1 -10906.869,E2 -10906.869} C_VEL
LIN {X 0,Y 409.398,Z 310.108,A -85,B 0,C 180,E1 -10907.483,E2 -10907.483} C_VEL
LIN {X 0,Y 410.05,Z 296.897,A -85,B 0,C 180,E1 -10907.905,E2 -10907.905} C_VEL
LIN {X 0,Y 411.038,Z 217.132,A -85,B 0,C 180,E1 -10909.365,E2 -10909.365} C_VEL
LIN {X 0,Y 408.12,Z 198.58,A -85,B 0,C 180,E1 -10909.882,E2 -10909.882} C_VEL
LIN {X 0,Y 406.199,Z 188.42,A -85,B 0,C 180,E1 -10910.201,E2 -10910.201} C_VEL
LIN {X 0,Y 407.649,Z 169.812,A -85,B 0,C 180,E1 -10913.972,E2 -10913.972} C_VEL
LIN {X 0,Y 407.683,Z 165,A -85,B 0,C 180,E1 -10914.983,E2 -10914.983} C_VEL
LIN {X 0,Y 405.7,Z 154.828,A -85,B 0,C 180,E1 -10917.3,E2 -10917.3} C_VEL
LIN {X 0,Y 404.186,Z 148.144,A -85,B 0,C 180,E1 -10918.921,E2 -10918.921} C_VEL
LIN {X 0,Y 404.142,Z 148.143,A -85,B 0,C 180,E1 -10922.622,E2 -10922.622} C_VEL
LIN {X 0,Y 404.177,Z 148.137,A -85,B 0,C 180,E1 -10925.188,E2 -10925.188} C_VEL
LIN {X 0,Y 404.136,Z 148.145,A -85,B 0,C 180,E1 -10928.759,E2 -10928.759} C_VEL
LIN {X 0,Y 404.108,Z 148.144,A -85,B 0,C 180,E1 -10931.597,E2 -10931.597} C_VEL
LIN {X 0,Y 404.146,Z 148.14,A -85,B 0,C 180,E1 -10934.521,E2 -10934.521} C_VEL
LIN {X 0,Y 404.122,Z 148.148,A -85,B 0,C 180,E1 -10937.293,E2 -10937.293} C_VEL
LIN {X 0,Y 404.135,Z 148.141,A -85,B 0,C 180,E1 -10939.951,E2 -10939.951} C_VEL
LIN {X 0,Y 404.132,Z 148.146,A -85,B 0,C 180,E1 -10943.126,E2 -10943.126} C_VEL
LIN {X 0,Y 404.138,Z 148.138,A -85,B 0,C 180,E1 -10946.186,E2 -10946.186} C_VEL
LIN {X 0,Y 404.141,Z 148.136,A -85,B 0,C 180,E1 -10949.714,E2 -10949.714} C_VEL
LIN {X 0,Y 404.099,Z 148.141,A -85,B 0,C 180,E1 -10953.115,E2 -10953.115} C_VEL
LIN {X 0,Y 404.148,Z 148.139,A -85,B 0,C 180,E1 -10956.424,E2 -10956.424} C_VEL
LIN {X 0,Y 404.15,Z 148.141,A -85,B 0,C 180,E1 -10959.891,E2 -10959.891} C_VEL
LIN {X 0,Y 404.157,Z 148.136,A -85,B 0,C 180,E1 -10963.021,E2 -10963.021} C_VEL
LIN {X 0,Y 404.286,Z 148.114,A -85,B 0,C 180,E1 -10966.938,E2 -10966.938} C_VEL
LIN {X 0,Y 404.249,Z 148.13,A -85,B 0,C 180,E1 -10969.988,E2 -10969.988} C_VEL
LIN {X 0,Y 404.344,Z 148.112,A -85,B 0,C 180,E1 -10973.011,E2 -10973.011} C_VEL
LIN {X 0,Y 404.264,Z 148.124,A -85,B 0,C 180,E1 -10975.013,E2 -10975.013} C_VEL
LIN {X 0,Y 404.474,Z 148.101,A -85,B 0,C 180,E1 -10978.008,E2 -10978.008} C_VEL
LIN {X 0,Y 404.353,Z 148.11,A -85,B 0,C 180,E1 -10980.995,E2 -10980.995} C_VEL
LIN {X 0,Y 404.408,Z 148.106,A -85,B 0,C 180,E1 -10982.988,E2 -10982.988} C_VEL
LIN {X 0,Y 404.348,Z 148.109,A -85,B 0,C 180,E1 -10986.511,E2 -10986.511} C_VEL
LIN {X 0,Y 404.268,Z 148.128,A -85,B 0,C 180,E1 -10989.001,E2 -10989.001} C_VEL
LIN {X 0,Y 404.258,Z 148.127,A -85,B 0,C 180,E1 -10992.041,E2 -10992.041} C_VEL
LIN {X 0,Y 404.207,Z 148.132,A -85,B 0,C 180,E1 -10995.117,E2 -10995.117} C_VEL
LIN {X 0,Y 404.205,Z 148.13,A -85,B 0,C 180,E1 -10998.238,E2 -10998.238} C_VEL
LIN {X 0,Y 404.139,Z 148.139,A -85,B 0,C 180,E1 -11001.419,E2 -11001.419} C_VEL
LIN {X 0,Y 404.17,Z 148.141,A -85,B 0,C 180,E1 -11004.665,E2 -11004.665} C_VEL
LIN {X 0,Y 404.195,Z 148.134,A -85,B 0,C 180,E1 -11007.999,E2 -11007.999} C_VEL
LIN {X 0,Y 404.138,Z 148.143,A -85,B 0,C 180,E1 -11011.557,E2 -11011.557} C_VEL
LIN {X 0,Y 404.183,Z 148.14,A -85,B 0,C 180,E1 -11015.016,E2 -11015.016} C_VEL
LIN {X 0,Y 404.153,Z 148.141,A -85,B 0,C 180,E1 -11018.756,E2 -11018.756} C_VEL
LIN {X 0,Y 404.121,Z 148.149,A -85,B 0,C 180,E1 -11021.599,E2 -11021.599} C_VEL
LIN {X 0,Y 404.143,Z 148.145,A -85,B 0,C 180,E1 -11024.522,E2 -11024.522} C_VEL
LIN {X 0,Y 404.172,Z 148.27,A -85,B 0,C 180,E1 -11026.438,E2 -11026.438} C_VEL
LIN {X 0,Y 406.416,Z 158.727,A -85,B 0,C 180,E1 -11029.115,E2 -11029.115} C_VEL
LIN {X 0,Y 406.763,Z 162.029,A -85,B 0,C 180,E1 -11029.889,E2 -11029.889} C_VEL
LIN {X 0,Y 410.685,Z 178.259,A -85,B 0,C 180,E1 -11030.436,E2 -11030.436} C_VEL
LIN {X 0,Y 411.657,Z 183.831,A -85,B 0,C 180,E1 -11030.599,E2 -11030.599} C_VEL
LIN {X 0,Y 410.282,Z 269.544,A -85,B 0,C 180,E1 -11032.16,E2 -11032.16} C_VEL
LIN {X 0,Y 409.838,Z 282.13,A -85,B 0,C 180,E1 -11032.577,E2 -11032.577} C_VEL
LIN {X 0,Y 409.28,Z 294.733,A -85,B 0,C 180,E1 -11033.197,E2 -11033.197} C_VEL
LIN {X 0,Y 408.524,Z 306.195,A -85,B 0,C 180,E1 -11033.954,E2 -11033.954} C_VEL
LIN {X 0,Y 407.669,Z 317.009,A -85,B 0,C 180,E1 -11034.875,E2 -11034.875} C_VEL
LIN {X 0,Y 406.756,Z 327.823,A -85,B 0,C 180,E1 -11036.031,E2 -11036.031} C_VEL
LIN {X 0,Y 405.953,Z 337.011,A -85,B 0,C 180,E1 -11037.247,E2 -11037.247} C_VEL
LIN {X 0,Y 405.125,Z 345.534,A -85,B 0,C 180,E1 -11038.639,E2 -11038.639} C_VEL
LIN {X 0,Y 404.454,Z 352.761,A -85,B 0,C 180,E1 -11040.099,E2 -11040.099} C_VEL
LIN {X 0,Y 403.95,Z 358.089,A -85,B 0,C 180,E1 -11041.416,E2 -11041.416} C_VEL
LIN {X 0,Y 403.527,Z 363.405,A -85,B 0,C 180,E1 -11043.075,E2 -11043.075} C_VEL
LIN {X 0,Y 403.292,Z 366.211,A -85,B 0,C 180,E1 -11044.172,E2 -11044.172} C_VEL
LIN {X 0,Y 403.108,Z 368.408,A -85,B 0,C 180,E1 -11045.265,E2 -11045.265} C_VEL
LIN {X 0,Y 402.939,Z 370.116,A -85,B 0,C 180,E1 -11046.349,E2 -11046.349} C_VEL
LIN {X 0,Y 402.852,Z 371.477,A -85,B 0,C 180,E1 -11047.609,E2 -11047.609} C_VEL
LIN {X 0,Y 402.729,Z 372.358,A -85,B 0,C 180,E1 -11049.573,E2 -11049.573} C_VEL
LIN {X 0,Y 402.755,Z 372.207,A -85,B 0,C 180,E1 -11050.637,E2 -11050.637} C_VEL
LIN {X 0,Y 402.749,Z 371.585,A -85,B 0,C 180,E1 -11051.693,E2 -11051.693} C_VEL
LIN {X 0,Y 402.922,Z 369.365,A -85,B 0,C 180,E1 -11053.603,E2 -11053.603} C_VEL
LIN {X 0,Y 403.135,Z 365.972,A -85,B 0,C 180,E1 -11055.358,E2 -11055.358} C_VEL
LIN {X 0,Y 403.395,Z 361.773,A -85,B 0,C 180,E1 -11056.91,E2 -11056.91} C_VEL
LIN {X 0,Y 403.701,Z 356.369,A -85,B 0,C 180,E1 -11058.451,E2 -11058.451} C_VEL
LIN {X 0,Y 404.199,Z 349.573,A -85,B 0,C 180,E1 -11059.987,E2 -11059.987} C_VEL
LIN {X 0,Y 404.745,Z 341.455,A -85,B 0,C 180,E1 -11061.463,E2 -11061.463} C_VEL
LIN {X 0,Y 405.441,Z 332.454,A -85,B 0,C 180,E1 -11062.78,E2 -11062.78} C_VEL
LIN {X 0,Y 406.242,Z 321.706,A -85,B 0,C 180,E1 -11064.042,E2 -11064.042} C_VEL
LIN {X 0,Y 406.995,Z 311.015,A -85,B 0,C 180,E1 -11065.047,E2 -11065.047} C_VEL
LIN {X 0,Y 407.59,Z 299.178,A -85,B 0,C 180,E1 -11065.921,E2 -11065.921} C_VEL
LIN {X 0,Y 407.822,Z 294.631,A -85,B 0,C 180,E1 -11066.2,E2 -11066.2} C_VEL
LIN {X 0,Y 407.274,Z 289.183,A -85,B 0,C 180,E1 -11066.523,E2 -11066.523} C_VEL
LIN {X 0,Y 403.701,Z 276.658,A -85,B 0,C 180,E1 -11067.203,E2 -11067.203} C_VEL
LIN {X 0,Y 402.115,Z 269.22,A -85,B 0,C 180,E1 -11067.494,E2 -11067.494} C_VEL
LIN {X 0,Y 401.902,Z 265.367,A -85,B 0,C 180,E1 -11067.593,E2 -11067.593} C_VEL
LIN {X 0,Y 402.924,Z 182.421,A -85,B 0,C 180,E1 -11069.097,E2 -11069.097} C_VEL
LIN {X 0,Y 398.978,Z 161.674,A -85,B 0,C 180,E1 -11069.669,E2 -11069.669} C_VEL
LIN {X 0,Y 398.927,Z 158.126,A -85,B 0,C 180,E1 -11070.505,E2 -11070.505} C_VEL
LIN {X 0,Y 397.38,Z 148.99,A -85,B 0,C 180,E1 -11072.788,E2 -11072.788} C_VEL
LIN {X 0,Y 397.314,Z 148.995,A -85,B 0,C 180,E1 -11076.093,E2 -11076.093} C_VEL
LIN {X 0,Y 397.222,Z 149.002,A -85,B 0,C 180,E1 -11079.163,E2 -11079.163} C_VEL
LIN {X 0,Y 397.203,Z 149.006,A -85,B 0,C 180,E1 -11082.259,E2 -11082.259} C_VEL
LIN {X 0,Y 397.105,Z 149.02,A -85,B 0,C 180,E1 -11085.395,E2 -11085.395} C_VEL
LIN {X 0,Y 397.08,Z 149.019,A -85,B 0,C 180,E1 -11088.578,E2 -11088.578} C_VEL
LIN {X 0,Y 397.082,Z 149.023,A -85,B 0,C 180,E1 -11091.82,E2 -11091.82} C_VEL
LIN {X 0,Y 397.096,Z 149.02,A -85,B 0,C 180,E1 -11095.136,E2 -11095.136} C_VEL
LIN {X 0,Y 397.056,Z 149.022,A -85,B 0,C 180,E1 -11098.549,E2 -11098.549} C_VEL
LIN {X 0,Y 397.071,Z 149.022,A -85,B 0,C 180,E1 -11101.835,E2 -11101.835} C_VEL
LIN {X 0,Y 397.112,Z 149.016,A -85,B 0,C 180,E1 -11104.495,E2 -11104.495} C_VEL
LIN {X 0,Y 397.086,Z 149.019,A -85,B 0,C 180,E1 -11108.277,E2 -11108.277} C_VEL
LIN {X 0,Y 397.049,Z 149.023,A -85,B 0,C 180,E1 -11111.977,E2 -11111.977} C_VEL
LIN {X 0,Y 397.084,Z 149.024,A -85,B 0,C 180,E1 -11115.07,E2 -11115.07} C_VEL
LIN {X 0,Y 397.05,Z 149.023,A -85,B 0,C 180,E1 -11118.025,E2 -11118.025} C_VEL
LIN {X 0,Y 397.089,Z 149.018,A -85,B 0,C 180,E1 -11121.724,E2 -11121.724} C_VEL
LIN {X 0,Y 397.115,Z 149.015,A -85,B 0,C 180,E1 -11125.506,E2 -11125.506} C_VEL
LIN {X 0,Y 397.071,Z 149.022,A -85,B 0,C 180,E1 -11129.118,E2 -11129.118} C_VEL
LIN {X 0,Y 397.058,Z 149.026,A -85,B 0,C 180,E1 -11132.254,E2 -11132.254} C_VEL
LIN {X 0,Y 397.102,Z 149.019,A -85,B 0,C 180,E1 -11134.865,E2 -11134.865} C_VEL
LIN {X 0,Y 397.088,Z 149.023,A -85,B 0,C 180,E1 -11138.182,E2 -11138.182} C_VEL
LIN {X 0,Y 397.084,Z 149.019,A -85,B 0,C 180,E1 -11141.423,E2 -11141.423} C_VEL
LIN {X 0,Y 397.112,Z 149.018,A -85,B 0,C 180,E1 -11144.606,E2 -11144.606} C_VEL
LIN {X 0,Y 397.21,Z 149.006,A -85,B 0,C 180,E1 -11147.742,E2 -11147.742} C_VEL
LIN {X 0,Y 397.23,Z 149.001,A -85,B 0,C 180,E1 -11150.838,E2 -11150.838} C_VEL
LIN {X 0,Y 397.323,Z 148.995,A -85,B 0,C 180,E1 -11153.908,E2 -11153.908} C_VEL
LIN {X 0,Y 397.442,Z 148.98,A -85,B 0,C 180,E1 -11157.974,E2 -11157.974} C_VEL
LIN {X 0,Y 397.444,Z 148.978,A -85,B 0,C 180,E1 -11162.027,E2 -11162.027} C_VEL
LIN {X 0,Y 397.322,Z 148.992,A -85,B 0,C 180,E1 -11166.093,E2 -11166.093} C_VEL
LIN {X 0,Y 397.234,Z 149.002,A -85,B 0,C 180,E1 -11169.163,E2 -11169.163} C_VEL
LIN {X 0,Y 397.224,Z 149.002,A -85,B 0,C 180,E1 -11172.258,E2 -11172.258} C_VEL
LIN {X 0,Y 397.129,Z 149.019,A -85,B 0,C 180,E1 -11175.395,E2 -11175.395} C_VEL
LIN {X 0,Y 397.119,Z 149.015,A -85,B 0,C 180,E1 -11178.576,E2 -11178.576} C_VEL
LIN {X 0,Y 397.098,Z 149.018,A -85,B 0,C 180,E1 -11181.819,E2 -11181.819} C_VEL
LIN {X 0,Y 397.107,Z 149.022,A -85,B 0,C 180,E1 -11185.135,E2 -11185.135} C_VEL
LIN {X 0,Y 397.067,Z 149.022,A -85,B 0,C 180,E1 -11188.549,E2 -11188.549} C_VEL
LIN {X 0,Y 397.082,Z 149.019,A -85,B 0,C 180,E1 -11191.835,E2 -11191.835} C_VEL
LIN {X 0,Y 397.122,Z 149.016,A -85,B 0,C 180,E1 -11194.494,E2 -11194.494} C_VEL
LIN {X 0,Y 397.098,Z 149.018,A -85,B 0,C 180,E1 -11198.276,E2 -11198.276} C_VEL
LIN {X 0,Y 397.056,Z 149.022,A -85,B 0,C 180,E1 -11201.976,E2 -11201.976} C_VEL
LIN {X 0,Y 397.089,Z 149.021,A -85,B 0,C 180,E1 -11205.069,E2 -11205.069} C_VEL
LIN {X 0,Y 397.056,Z 149.023,A -85,B 0,C 180,E1 -11208.024,E2 -11208.024} C_VEL
LIN {X 0,Y 397.096,Z 149.017,A -85,B 0,C 180,E1 -11211.724,E2 -11211.724} C_VEL
LIN {X 0,Y 397.123,Z 149.014,A -85,B 0,C 180,E1 -11215.506,E2 -11215.506} C_VEL
LIN {X 0,Y 397.081,Z 149.023,A -85,B 0,C 180,E1 -11219.117,E2 -11219.117} C_VEL
LIN {X 0,Y 397.18,Z 149.052,A -85,B 0,C 180,E1 -11222.003,E2 -11222.003} C_VEL
LIN {X 0,Y 400.043,Z 164.134,A -85,B 0,C 180,E1 -11225.336,E2 -11225.336} C_VEL
LIN {X 0,Y 399.474,Z 174.742,A -85,B 0,C 180,E1 -11227.502,E2 -11227.502} C_VEL
LIN {X 0,Y 398.544,Z 188.839,A -85,B 0,C 180,E1 -11230.34,E2 -11230.34} C_VEL
LIN {X 0,Y 402.673,Z 218.907,A -85,B 0,C 180,E1 -11231.076,E2 -11231.076} C_VEL
LIN {X 0,Y 401.643,Z 297.984,A -85,B 0,C 180,E1 -11232.53,E2 -11232.53} C_VEL
LIN {X 0,Y 401.061,Z 311.755,A -85,B 0,C 180,E1 -11232.997,E2 -11232.997} C_VEL
LIN {X 0,Y 400.425,Z 324.157,A -85,B 0,C 180,E1 -11233.625,E2 -11233.625} C_VEL
LIN {X 0,Y 399.625,Z 336.048,A -85,B 0,C 180,E1 -11234.443,E2 -11234.443} C_VEL
LIN {X 0,Y 398.859,Z 347.504,A -85,B 0,C 180,E1 -11235.458,E2 -11235.458} C_VEL
LIN {X 0,Y 398.194,Z 357.397,A -85,B 0,C 180,E1 -11236.551,E2 -11236.551} C_VEL
LIN {X 0,Y 397.546,Z 366.267,A -85,B 0,C 180,E1 -11237.752,E2 -11237.752} C_VEL
LIN {X 0,Y 396.786,Z 375.407,A -85,B 0,C 180,E1 -11239.281,E2 -11239.281} C_VEL
LIN {X 0,Y 396.335,Z 382.775,A -85,B 0,C 180,E1 -11240.817,E2 -11240.817} C_VEL
LIN {X 0,Y 396.044,Z 388.671,A -85,B 0,C 180,E1 -11242.351,E2 -11242.351} C_VEL
LIN {X 0,Y 395.822,Z 394.096,A -85,B 0,C 180,E1 -11244.204,E2 -11244.204} C_VEL
LIN {X 0,Y 395.779,Z 397.733,A -85,B 0,C 180,E1 -11245.927,E2 -11245.927} C_VEL
LIN {X 0,Y 395.748,Z 399.304,A -85,B 0,C 180,E1 -11246.946,E2 -11246.946} C_VEL
LIN {X 0,Y 395.823,Z 400.444,A -85,B 0,C 180,E1 -11247.965,E2 -11247.965} C_VEL
LIN {X 0,Y 395.812,Z 401.15,A -85,B 0,C 180,E1 -11248.982,E2 -11248.982} C_VEL
LIN {X 0,Y 395.8,Z 401.466,A -85,B 0,C 180,E1 -11250,E2 -11250} C_VEL
LIN {X 0,Y 395.797,Z 401.393,A -85,B 0,C 180,E1 -11251.017,E2 -11251.017} C_VEL
LIN {X 0,Y 395.804,Z 400.915,A -85,B 0,C 180,E1 -11252.035,E2 -11252.035} C_VEL
LIN {X 0,Y 395.775,Z 398.703,A -85,B 0,C 180,E1 -11254.073,E2 -11254.073} C_VEL
LIN {X 0,Y 395.797,Z 395.624,A -85,B 0,C 180,E1 -11255.761,E2 -11255.761} C_VEL
LIN {X 0,Y 396.064,Z 390.716,A -85,B 0,C 180,E1 -11257.648,E2 -11257.648} C_VEL
LIN {X 0,Y 396.492,Z 384.425,A -85,B 0,C 180,E1 -11259.437,E2 -11259.437} C_VEL
LIN {X 0,Y 397.009,Z 377.596,A -85,B 0,C 180,E1 -11260.97,E2 -11260.97} C_VEL
LIN {X 0,Y 397.957,Z 369.119,A -85,B 0,C 180,E1 -11262.494,E2 -11262.494} C_VEL
LIN {X 0,Y 398.775,Z 359.221,A -85,B 0,C 180,E1 -11263.923,E2 -11263.923} C_VEL
LIN {X 0,Y 399.741,Z 348.671,A -85,B 0,C 180,E1 -11265.147,E2 -11265.147} C_VEL
LIN {X 0,Y 400.729,Z 337.577,A -85,B 0,C 180,E1 -11266.166,E2 -11266.166} C_VEL
LIN {X 0,Y 401.748,Z 325.309,A -85,B 0,C 180,E1 -11267.039,E2 -11267.039} C_VEL
LIN {X 0,Y 402.581,Z 312.411,A -85,B 0,C 180,E1 -11267.723,E2 -11267.723} C_VEL
LIN {X 0,Y 403.3,Z 299.375,A -85,B 0,C 180,E1 -11268.182,E2 -11268.182} C_VEL
LIN {X 0,Y 403.706,Z 278.729,A -85,B 0,C 180,E1 -11268.605,E2 -11268.605} C_VEL
LIN {X 0,Y 404.449,Z 217.875,A -85,B 0,C 180,E1 -11269.729,E2 -11269.729} C_VEL
LIN {X 0,Y 401.509,Z 199.352,A -85,B 0,C 180,E1 -11270.263,E2 -11270.263} C_VEL
LIN {X 0,Y 399.355,Z 188.093,A -85,B 0,C 180,E1 -11270.636,E2 -11270.636} C_VEL
LIN {X 0,Y 400.817,Z 170.585,A -85,B 0,C 180,E1 -11274.247,E2 -11274.247} C_VEL
LIN {X 0,Y 400.76,Z 166.314,A -85,B 0,C 180,E1 -11275.167,E2 -11275.167} C_VEL
LIN {X 0,Y 398.713,Z 156.068,A -85,B 0,C 180,E1 -11277.558,E2 -11277.558} C_VEL
LIN {X 0,Y 397.131,Z 149.024,A -85,B 0,C 180,E1 -11279.303,E2 -11279.303} C_VEL
LIN {X 0,Y 397.115,Z 149.023,A -85,B 0,C 180,E1 -11283.273,E2 -11283.273} C_VEL
LIN {X 0,Y 397.108,Z 149.021,A -85,B 0,C 180,E1 -11285.735,E2 -11285.735} C_VEL
LIN {X 0,Y 397.094,Z 149.023,A -85,B 0,C 180,E1 -11288.854,E2 -11288.854} C_VEL
LIN {X 0,Y 397.056,Z 149.025,A -85,B 0,C 180,E1 -11292.269,E2 -11292.269} C_VEL
LIN {X 0,Y 397.088,Z 149.024,A -85,B 0,C 180,E1 -11295.069,E2 -11295.069} C_VEL
LIN {X 0,Y 397.053,Z 149.025,A -85,B 0,C 180,E1 -11298.024,E2 -11298.024} C_VEL
LIN {X 0,Y 397.09,Z 149.017,A -85,B 0,C 180,E1 -11301.723,E2 -11301.723} C_VEL
LIN {X 0,Y 397.117,Z 149.012,A -85,B 0,C 180,E1 -11305.505,E2 -11305.505} C_VEL
LIN {X 0,Y 397.073,Z 149.017,A -85,B 0,C 180,E1 -11309.116,E2 -11309.116} C_VEL
LIN {X 0,Y 397.06,Z 149.024,A -85,B 0,C 180,E1 -11312.253,E2 -11312.253} C_VEL
LIN {X 0,Y 397.104,Z 149.019,A -85,B 0,C 180,E1 -11314.864,E2 -11314.864} C_VEL
LIN {X 0,Y 397.089,Z 149.015,A -85,B 0,C 180,E1 -11318.181,E2 -11318.181} C_VEL
LIN {X 0,Y 397.087,Z 149.016,A -85,B 0,C 180,E1 -11321.422,E2 -11321.422} C_VEL
LIN {X 0,Y 397.126,Z 149.017,A -85,B 0,C 180,E1 -11324.605,E2 -11324.605} C_VEL
LIN {X 0,Y 397.217,Z 148.998,A -85,B 0,C 180,E1 -11327.741,E2 -11327.741} C_VEL
LIN {X 0,Y 397.232,Z 148.997,A -85,B 0,C 180,E1 -11330.837,E2 -11330.837} C_VEL
LIN {X 0,Y 397.331,Z 148.993,A -85,B 0,C 180,E1 -11333.907,E2 -11333.907} C_VEL
LIN {X 0,Y 397.442,Z 148.976,A -85,B 0,C 180,E1 -11337.973,E2 -11337.973} C_VEL
LIN {X 0,Y 397.323,Z 148.986,A -85,B 0,C 180,E1 -11341.013,E2 -11341.013} C_VEL
LIN {X 0,Y 397.368,Z 148.983,A -85,B 0,C 180,E1 -11343.041,E2 -11343.041} C_VEL
LIN {X 0,Y 397.304,Z 148.987,A -85,B 0,C 180,E1 -11346.504,E2 -11346.504} C_VEL
LIN {X 0,Y 397.237,Z 149.004,A -85,B 0,C 180,E1 -11349.162,E2 -11349.162} C_VEL
LIN {X 0,Y 397.221,Z 149.003,A -85,B 0,C 180,E1 -11352.257,E2 -11352.257} C_VEL
LIN {X 0,Y 397.18,Z 149.009,A -85,B 0,C 180,E1 -11355.391,E2 -11355.391} C_VEL
LIN {X 0,Y 397.159,Z 149.008,A -85,B 0,C 180,E1 -11358.573,E2 -11358.573} C_VEL
LIN {X 0,Y 397.096,Z 149.014,A -85,B 0,C 180,E1 -11361.818,E2 -11361.818} C_VEL
LIN {X 0,Y 397.151,Z 149.013,A -85,B 0,C 180,E1 -11365.511,E2 -11365.511} C_VEL
LIN {X 0,Y 397.122,Z 149.018,A -85,B 0,C 180,E1 -11368.543,E2 -11368.543} C_VEL
LIN {X 0,Y 397.077,Z 149.024,A -85,B 0,C 180,E1 -11372.071,E2 -11372.071} C_VEL
LIN {X 0,Y 397.118,Z 149.019,A -85,B 0,C 180,E1 -11375.503,E2 -11375.503} C_VEL
LIN {X 0,Y 397.128,Z 149.015,A -85,B 0,C 180,E1 -11378.861,E2 -11378.861} C_VEL
LIN {X 0,Y 397.067,Z 149.028,A -85,B 0,C 180,E1 -11382.267,E2 -11382.267} C_VEL
LIN {X 0,Y 397.085,Z 149.025,A -85,B 0,C 180,E1 -11385.068,E2 -11385.068} C_VEL
LIN {X 0,Y 397.124,Z 149.168,A -85,B 0,C 180,E1 -11386.086,E2 -11386.086} C_VEL
LIN {X 0,Y 399.613,Z 160.87,A -85,B 0,C 180,E1 -11389.133,E2 -11389.133} C_VEL
LIN {X 0,Y 399.836,Z 162.319,A -85,B 0,C 180,E1 -11389.461,E2 -11389.461} C_VEL
LIN {X 0,Y 402.585,Z 172.468,A -85,B 0,C 180,E1 -11389.832,E2 -11389.832} C_VEL
LIN {X 0,Y 405.117,Z 184.576,A -85,B 0,C 180,E1 -11390.223,E2 -11390.223} C_VEL
LIN {X 0,Y 403.67,Z 269.169,A -85,B 0,C 180,E1 -11391.786,E2 -11391.786} C_VEL
LIN {X 0,Y 403.206,Z 281.839,A -85,B 0,C 180,E1 -11392.205,E2 -11392.205} C_VEL
LIN {X 0,Y 402.644,Z 294.226,A -85,B 0,C 180,E1 -11392.817,E2 -11392.817} C_VEL
LIN {X 0,Y 401.894,Z 305.403,A -85,B 0,C 180,E1 -11393.552,E2 -11393.552} C_VEL
LIN {X 0,Y 400.965,Z 316.661,A -85,B 0,C 180,E1 -11394.507,E2 -11394.507} C_VEL
LIN {X 0,Y 400.018,Z 327.419,A -85,B 0,C 180,E1 -11395.664,E2 -11395.664} C_VEL
LIN {X 0,Y 399.114,Z 336.835,A -85,B 0,C 180,E1 -11396.915,E2 -11396.915} C_VEL
LIN {X 0,Y 398.246,Z 345.469,A -85,B 0,C 180,E1 -11398.331,E2 -11398.331} C_VEL
LIN {X 0,Y 397.605,Z 352.122,A -85,B 0,C 180,E1 -11399.671,E2 -11399.671} C_VEL
LIN {X 0,Y 396.883,Z 359.121,A -85,B 0,C 180,E1 -11401.438,E2 -11401.438} C_VEL
LIN {X 0,Y 396.433,Z 364.27,A -85,B 0,C 180,E1 -11403.124,E2 -11403.124} C_VEL
LIN {X 0,Y 396.094,Z 368.099,A -85,B 0,C 180,E1 -11404.809,E2 -11404.809} C_VEL
LIN {X 0,Y 395.905,Z 369.908,A -85,B 0,C 180,E1 -11405.903,E2 -11405.903} C_VEL
LIN {X 0,Y 395.783,Z 371.664,A -85,B 0,C 180,E1 -11407.423,E2 -11407.423} C_VEL
LIN {X 0,Y 395.657,Z 372.572,A -85,B 0,C 180,E1 -11409.191,E2 -11409.191} C_VEL
LIN {X 0,Y 395.661,Z 372.545,A -85,B 0,C 180,E1 -11410.29,E2 -11410.29} C_VEL
LIN {X 0,Y 395.67,Z 372.097,A -85,B 0,C 180,E1 -11411.354,E2 -11411.354} C_VEL
LIN {X 0,Y 395.69,Z 371.166,A -85,B 0,C 180,E1 -11412.426,E2 -11412.426} C_VEL
LIN {X 0,Y 395.816,Z 369.806,A -85,B 0,C 180,E1 -11413.496,E2 -11413.496} C_VEL
LIN {X 0,Y 396.021,Z 366.918,A -85,B 0,C 180,E1 -11415.089,E2 -11415.089} C_VEL
LIN {X 0,Y 396.279,Z 362.954,A -85,B 0,C 180,E1 -11416.67,E2 -11416.67} C_VEL
LIN {X 0,Y 396.584,Z 357.823,A -85,B 0,C 180,E1 -11418.241,E2 -11418.241} C_VEL
LIN {X 0,Y 397.03,Z 351.351,A -85,B 0,C 180,E1 -11419.804,E2 -11419.804} C_VEL
LIN {X 0,Y 397.643,Z 343.088,A -85,B 0,C 180,E1 -11421.384,E2 -11421.384} C_VEL
LIN {X 0,Y 398.334,Z 334.928,A -85,B 0,C 180,E1 -11422.651,E2 -11422.651} C_VEL
LIN {X 0,Y 399.107,Z 324.805,A -85,B 0,C 180,E1 -11423.935,E2 -11423.935} C_VEL
LIN {X 0,Y 399.83,Z 314.749,A -85,B 0,C 180,E1 -11424.958,E2 -11424.958} C_VEL
LIN {X 0,Y 400.508,Z 303.82,A -85,B 0,C 180,E1 -11425.849,E2 -11425.849} C_VEL
LIN {X 0,Y 401.027,Z 292.06,A -85,B 0,C 180,E1 -11426.597,E2 -11426.597} C_VEL
LIN {X 0,Y 401.522,Z 279.577,A -85,B 0,C 180,E1 -11427.178,E2 -11427.178} C_VEL
LIN {X 0,Y 401.883,Z 267.023,A -85,B 0,C 180,E1 -11427.557,E2 -11427.557} C_VEL
LIN {X 0,Y 401.902,Z 265.367,A -85,B 0,C 180,E1 -11427.593,E2 -11427.593} C_VEL
LIN {X 0,Y 401.357,Z 259.562,A -85,B 0,C 180,E1 -11427.735,E2 -11427.735} C_VEL
LIN {X 0,Y 395.959,Z 240.852,A -85,B 0,C 180,E1 -11428.299,E2 -11428.299} C_VEL
LIN {X 0,Y 395.47,Z 235.033,A -85,B 0,C 180,E1 -11428.426,E2 -11428.426} C_VEL
LIN {X 0,Y 396.196,Z 183.667,A -85,B 0,C 180,E1 -11429.365,E2 -11429.365} C_VEL
LIN {X 0,Y 392.046,Z 161.932,A -85,B 0,C 180,E1 -11429.971,E2 -11429.971} C_VEL
LIN {X 0,Y 391.807,Z 158.622,A -85,B 0,C 180,E1 -11430.771,E2 -11430.771} C_VEL
LIN {X 0,Y 390.284,Z 149.874,A -85,B 0,C 180,E1 -11432.968,E2 -11432.968} C_VEL
LIN {X 0,Y 390.27,Z 149.871,A -85,B 0,C 180,E1 -11436.203,E2 -11436.203} C_VEL
LIN {X 0,Y 390.181,Z 149.88,A -85,B 0,C 180,E1 -11439.33,E2 -11439.33} C_VEL
LIN {X 0,Y 390.149,Z 149.883,A -85,B 0,C 180,E1 -11442.484,E2 -11442.484} C_VEL
LIN {X 0,Y 390.049,Z 149.902,A -85,B 0,C 180,E1 -11445.681,E2 -11445.681} C_VEL
LIN {X 0,Y 390.037,Z 149.897,A -85,B 0,C 180,E1 -11448.926,E2 -11448.926} C_VEL
LIN {X 0,Y 390.025,Z 149.899,A -85,B 0,C 180,E1 -11452.235,E2 -11452.235} C_VEL
LIN {X 0,Y 390.047,Z 149.899,A -85,B 0,C 180,E1 -11455.723,E2 -11455.723} C_VEL
LIN {X 0,Y 390.018,Z 149.903,A -85,B 0,C 180,E1 -11459.113,E2 -11459.113} C_VEL
LIN {X 0,Y 390.035,Z 149.898,A -85,B 0,C 180,E1 -11462.723,E2 -11462.723} C_VEL
LIN {X 0,Y 390.038,Z 149.897,A -85,B 0,C 180,E1 -11465.823,E2 -11465.823} C_VEL
LIN {X 0,Y 390.033,Z 149.903,A -85,B 0,C 180,E1 -11469.213,E2 -11469.213} C_VEL
LIN {X 0,Y 390.027,Z 149.899,A -85,B 0,C 180,E1 -11472.373,E2 -11472.373} C_VEL
LIN {X 0,Y 390.039,Z 149.899,A -85,B 0,C 180,E1 -11475.355,E2 -11475.355} C_VEL
LIN {X 0,Y 390.013,Z 149.9,A -85,B 0,C 180,E1 -11478.185,E2 -11478.185} C_VEL
LIN {X 0,Y 390.056,Z 149.9,A -85,B 0,C 180,E1 -11480.904,E2 -11480.904} C_VEL
LIN {X 0,Y 390.068,Z 149.899,A -85,B 0,C 180,E1 -11484.792,E2 -11484.792} C_VEL
LIN {X 0,Y 390.017,Z 149.904,A -85,B 0,C 180,E1 -11488.496,E2 -11488.496} C_VEL
LIN {X 0,Y 390.016,Z 149.901,A -85,B 0,C 180,E1 -11492.004,E2 -11492.004} C_VEL
LIN {X 0,Y 390.041,Z 149.896,A -85,B 0,C 180,E1 -11495.517,E2 -11495.517} C_VEL
LIN {X 0,Y 390.049,Z 149.897,A -85,B 0,C 180,E1 -11498.878,E2 -11498.878} C_VEL
LIN {X 0,Y 390.072,Z 149.894,A -85,B 0,C 180,E1 -11502.731,E2 -11502.731} C_VEL
LIN {X 0,Y 390.135,Z 149.887,A -85,B 0,C 180,E1 -11506.601,E2 -11506.601} C_VEL
LIN {X 0,Y 390.159,Z 149.883,A -85,B 0,C 180,E1 -11509.623,E2 -11509.623} C_VEL
LIN {X 0,Y 390.25,Z 149.871,A -85,B 0,C 180,E1 -11512.758,E2 -11512.758} C_VEL
LIN {X 0,Y 390.202,Z 149.876,A -85,B 0,C 180,E1 -11514.834,E2 -11514.834} C_VEL
LIN {X 0,Y 390.408,Z 149.857,A -85,B 0,C 180,E1 -11517.937,E2 -11517.937} C_VEL
LIN {X 0,Y 390.411,Z 149.854,A -85,B 0,C 180,E1 -11522.064,E2 -11522.064} C_VEL
LIN {X 0,Y 390.278,Z 149.868,A -85,B 0,C 180,E1 -11526.203,E2 -11526.203} C_VEL
LIN {X 0,Y 390.193,Z 149.881,A -85,B 0,C 180,E1 -11529.33,E2 -11529.33} C_VEL
LIN {X 0,Y 390.176,Z 149.879,A -85,B 0,C 180,E1 -11532.483,E2 -11532.483} C_VEL
LIN {X 0,Y 390.072,Z 149.896,A -85,B 0,C 180,E1 -11535.68,E2 -11535.68} C_VEL
LIN {X 0,Y 390.076,Z 149.894,A -85,B 0,C 180,E1 -11538.924,E2 -11538.924} C_VEL
LIN {X 0,Y 390.039,Z 149.896,A -85,B 0,C 180,E1 -11542.235,E2 -11542.235} C_VEL
LIN {X 0,Y 390.055,Z 149.896,A -85,B 0,C 180,E1 -11545.722,E2 -11545.722} C_VEL
LIN {X 0,Y 390.029,Z 149.905,A -85,B 0,C 180,E1 -11549.113,E2 -11549.113} C_VEL
LIN {X 0,Y 390.044,Z 149.899,A -85,B 0,C 180,E1 -11552.722,E2 -11552.722} C_VEL
LIN {X 0,Y 390.048,Z 149.895,A -85,B 0,C 180,E1 -11555.823,E2 -11555.823} C_VEL
LIN {X 0,Y 390.043,Z 149.899,A -85,B 0,C 180,E1 -11559.213,E2 -11559.213} C_VEL
LIN {X 0,Y 390.034,Z 149.899,A -85,B 0,C 180,E1 -11562.372,E2 -11562.372} C_VEL
LIN {X 0,Y 390.045,Z 149.896,A -85,B 0,C 180,E1 -11565.354,E2 -11565.354} C_VEL
LIN {X 0,Y 390.019,Z 149.901,A -85,B 0,C 180,E1 -11568.184,E2 -11568.184} C_VEL
LIN {X 0,Y 390.062,Z 149.897,A -85,B 0,C 180,E1 -11570.904,E2 -11570.904} C_VEL
LIN {X 0,Y 390.085,Z 149.894,A -85,B 0,C 180,E1 -11574.793,E2 -11574.793} C_VEL
LIN {X 0,Y 390.027,Z 149.904,A -85,B 0,C 180,E1 -11578.495,E2 -11578.495} C_VEL
LIN {X 0,Y 390.11,Z 149.926,A -85,B 0,C 180,E1 -11581.766,E2 -11581.766} C_VEL
LIN {X 0,Y 393.028,Z 164.937,A -85,B 0,C 180,E1 -11585.151,E2 -11585.151} C_VEL
LIN {X 0,Y 392.785,Z 171.573,A -85,B 0,C 180,E1 -11586.539,E2 -11586.539} C_VEL
LIN {X 0,Y 391.596,Z 188.557,A -85,B 0,C 180,E1 -11590.028,E2 -11590.028} C_VEL
LIN {X 0,Y 395.879,Z 219.989,A -85,B 0,C 180,E1 -11590.813,E2 -11590.813} C_VEL
LIN {X 0,Y 394.805,Z 297.205,A -85,B 0,C 180,E1 -11592.251,E2 -11592.251} C_VEL
LIN {X 0,Y 394.278,Z 310.389,A -85,B 0,C 180,E1 -11592.695,E2 -11592.695} C_VEL
LIN {X 0,Y 393.552,Z 323.102,A -85,B 0,C 180,E1 -11593.331,E2 -11593.331} C_VEL
LIN {X 0,Y 392.782,Z 335.213,A -85,B 0,C 180,E1 -11594.165,E2 -11594.165} C_VEL
LIN {X 0,Y 391.924,Z 346.768,A -85,B 0,C 180,E1 -11595.195,E2 -11595.195} C_VEL
LIN {X 0,Y 391.219,Z 356.978,A -85,B 0,C 180,E1 -11596.336,E2 -11596.336} C_VEL
LIN {X 0,Y 390.545,Z 365.698,A -85,B 0,C 180,E1 -11597.529,E2 -11597.529} C_VEL
LIN {X 0,Y 389.763,Z 374.9,A -85,B 0,C 180,E1 -11599.086,E2 -11599.086} C_VEL
LIN {X 0,Y 389.288,Z 382.313,A -85,B 0,C 180,E1 -11600.649,E2 -11600.649} C_VEL
LIN {X 0,Y 388.976,Z 388.249,A -85,B 0,C 180,E1 -11602.212,E2 -11602.212} C_VEL
LIN {X 0,Y 388.775,Z 393.139,A -85,B 0,C 180,E1 -11603.857,E2 -11603.857} C_VEL
LIN {X 0,Y 388.715,Z 396.461,A -85,B 0,C 180,E1 -11605.333,E2 -11605.333} C_VEL
LIN {X 0,Y 388.653,Z 398.979,A -85,B 0,C 180,E1 -11606.89,E2 -11606.89} C_VEL
LIN {X 0,Y 388.721,Z 400.147,A -85,B 0,C 180,E1 -11607.928,E2 -11607.928} C_VEL
LIN {X 0,Y 388.742,Z 400.869,A -85,B 0,C 180,E1 -11608.964,E2 -11608.964} C_VEL
LIN {X 0,Y 388.729,Z 401.199,A -85,B 0,C 180,E1 -11610,E2 -11610} C_VEL
LIN {X 0,Y 388.728,Z 401.141,A -85,B 0,C 180,E1 -11611.036,E2 -11611.036} C_VEL
LIN {X 0,Y 388.701,Z 400.685,A -85,B 0,C 180,E1 -11612.072,E2 -11612.072} C_VEL
LIN {X 0,Y 388.699,Z 398.504,A -85,B 0,C 180,E1 -11614.147,E2 -11614.147} C_VEL
LIN {X 0,Y 388.733,Z 394.997,A -85,B 0,C 180,E1 -11616.085,E2 -11616.085} C_VEL
LIN {X 0,Y 389.018,Z 390.592,A -85,B 0,C 180,E1 -11617.787,E2 -11617.787} C_VEL
LIN {X 0,Y 389.471,Z 384.334,A -85,B 0,C 180,E1 -11619.608,E2 -11619.608} C_VEL
LIN {X 0,Y 390.019,Z 377.542,A -85,B 0,C 180,E1 -11621.169,E2 -11621.169} C_VEL
LIN {X 0,Y 391.011,Z 369.135,A -85,B 0,C 180,E1 -11622.72,E2 -11622.72} C_VEL
LIN {X 0,Y 391.826,Z 359.826,A -85,B 0,C 180,E1 -11624.106,E2 -11624.106} C_VEL
LIN {X 0,Y 392.882,Z 348.872,A -85,B 0,C 180,E1 -11625.418,E2 -11625.418} C_VEL
LIN {X 0,Y 393.929,Z 337.967,A -85,B 0,C 180,E1 -11626.453,E2 -11626.453} C_VEL
LIN {X 0,Y 394.992,Z 325.897,A -85,B 0,C 180,E1 -11627.339,E2 -11627.339} C_VEL
LIN {X 0,Y 395.867,Z 313.328,A -85,B 0,C 180,E1 -11628.034,E2 -11628.034} C_VEL
LIN {X 0,Y 396.582,Z 301.072,A -85,B 0,C 180,E1 -11628.501,E2 -11628.501} C_VEL
LIN {X 0,Y 396.986,Z 287.213,A -85,B 0,C 180,E1 -11628.821,E2 -11628.821} C_VEL
LIN {X 0,Y 397.862,Z 218.121,A -85,B 0,C 180,E1 -11630.119,E2 -11630.119} C_VEL
LIN {X 0,Y 394.167,Z 195.95,A -85,B 0,C 180,E1 -11630.788,E2 -11630.788} C_VEL
LIN {X 0,Y 392.522,Z 187.884,A -85,B 0,C 180,E1 -11631.06,E2 -11631.06} C_VEL
LIN {X 0,Y 393.994,Z 171.359,A -85,B 0,C 180,E1 -11634.531,E2 -11634.531} C_VEL
LIN {X 0,Y 393.848,Z 167.636,A -85,B 0,C 180,E1 -11635.358,E2 -11635.358} C_VEL
LIN {X 0,Y 391.501,Z 156.071,A -85,B 0,C 180,E1 -11638.132,E2 -11638.132} C_VEL
LIN {X 0,Y 390.074,Z 149.9,A -85,B 0,C 180,E1 -11639.701,E2 -11639.701} C_VEL
LIN {X 0,Y 390.044,Z 149.9,A -85,B 0,C 180,E1 -11642.721,E2 -11642.721} C_VEL
LIN {X 0,Y 390.055,Z 149.899,A -85,B 0,C 180,E1 -11645.824,E2 -11645.824} C_VEL
LIN {X 0,Y 390.039,Z 149.904,A -85,B 0,C 180,E1 -11649.212,E2 -11649.212} C_VEL
LIN {X 0,Y 390.032,Z 149.9,A -85,B 0,C 180,E1 -11652.372,E2 -11652.372} C_VEL
LIN {X 0,Y 390.043,Z 149.901,A -85,B 0,C 180,E1 -11655.354,E2 -11655.354} C_VEL
LIN {X 0,Y 390.016,Z 149.902,A -85,B 0,C 180,E1 -11658.184,E2 -11658.184} C_VEL
LIN {X 0,Y 390.058,Z 149.9,A -85,B 0,C 180,E1 -11660.903,E2 -11660.903} C_VEL
LIN {X 0,Y 390.069,Z 149.894,A -85,B 0,C 180,E1 -11664.791,E2 -11664.791} C_VEL
LIN {X 0,Y 390.018,Z 149.9,A -85,B 0,C 180,E1 -11668.495,E2 -11668.495} C_VEL
LIN {X 0,Y 390.017,Z 149.9,A -85,B 0,C 180,E1 -11672.003,E2 -11672.003} C_VEL
LIN {X 0,Y 390.042,Z 149.896,A -85,B 0,C 180,E1 -11675.516,E2 -11675.516} C_VEL
LIN {X 0,Y 390.049,Z 149.897,A -85,B 0,C 180,E1 -11678.877,E2 -11678.877} C_VEL
LIN {X 0,Y 390.073,Z 149.892,A -85,B 0,C 180,E1 -11682.729,E2 -11682.729} C_VEL
LIN {X 0,Y 390.198,Z 149.87,A -85,B 0,C 180,E1 -11686.561,E2 -11686.561} C_VEL
LIN {X 0,Y 390.19,Z 149.875,A -85,B 0,C 180,E1 -11690.67,E2 -11690.67} C_VEL
LIN {X 0,Y 390.285,Z 149.869,A -85,B 0,C 180,E1 -11693.797,E2 -11693.797} C_VEL
LIN {X 0,Y 390.409,Z 149.851,A -85,B 0,C 180,E1 -11697.936,E2 -11697.936} C_VEL
LIN {X 0,Y 390.294,Z 149.862,A -85,B 0,C 180,E1 -11701.031,E2 -11701.031} C_VEL
LIN {X 0,Y 390.302,Z 149.864,A -85,B 0,C 180,E1 -11703.096,E2 -11703.096} C_VEL
LIN {X 0,Y 390.264,Z 149.864,A -85,B 0,C 180,E1 -11706.495,E2 -11706.495} C_VEL
LIN {X 0,Y 390.195,Z 149.878,A -85,B 0,C 180,E1 -11709.328,E2 -11709.328} C_VEL
LIN {X 0,Y 390.172,Z 149.882,A -85,B 0,C 180,E1 -11712.482,E2 -11712.482} C_VEL
LIN {X 0,Y 390.14,Z 149.887,A -85,B 0,C 180,E1 -11715.676,E2 -11715.676} C_VEL
LIN {X 0,Y 390.103,Z 149.889,A -85,B 0,C 180,E1 -11718.922,E2 -11718.922} C_VEL
LIN {X 0,Y 390.037,Z 149.894,A -85,B 0,C 180,E1 -11722.234,E2 -11722.234} C_VEL
LIN {X 0,Y 390.117,Z 149.889,A -85,B 0,C 180,E1 -11725.742,E2 -11725.742} C_VEL
LIN {X 0,Y 390.058,Z 149.9,A -85,B 0,C 180,E1 -11729.109,E2 -11729.109} C_VEL
LIN {X 0,Y 390.042,Z 149.9,A -85,B 0,C 180,E1 -11732.721,E2 -11732.721} C_VEL
LIN {X 0,Y 390.054,Z 149.9,A -85,B 0,C 180,E1 -11735.825,E2 -11735.825} C_VEL
LIN {X 0,Y 390.068,Z 149.895,A -85,B 0,C 180,E1 -11739.218,E2 -11739.218} C_VEL
LIN {X 0,Y 390.04,Z 149.903,A -85,B 0,C 180,E1 -11742.374,E2 -11742.374} C_VEL
LIN {X 0,Y 390.075,Z 150.047,A -85,B 0,C 180,E1 -11745.701,E2 -11745.701} C_VEL
LIN {X 0,Y 392.582,Z 161.467,A -85,B 0,C 180,E1 -11748.753,E2 -11748.753} C_VEL
LIN {X 0,Y 392.797,Z 162.641,A -85,B 0,C 180,E1 -11749.009,E2 -11749.009} C_VEL
LIN {X 0,Y 395.423,Z 170.997,A -85,B 0,C 180,E1 -11749.349,E2 -11749.349} C_VEL
LIN {X 0,Y 398.52,Z 184.985,A -85,B 0,C 180,E1 -11749.824,E2 -11749.824} C_VEL
LIN {X 0,Y 397.084,Z 269.872,A -85,B 0,C 180,E1 -11751.428,E2 -11751.428} C_VEL
LIN {X 0,Y 396.561,Z 282.705,A -85,B 0,C 180,E1 -11751.865,E2 -11751.865} C_VEL
LIN {X 0,Y 395.907,Z 296.124,A -85,B 0,C 180,E1 -11752.555,E2 -11752.555} C_VEL
LIN {X 0,Y 395.039,Z 307.903,A -85,B 0,C 180,E1 -11753.384,E2 -11753.384} C_VEL
LIN {X 0,Y 394.022,Z 319.287,A -85,B 0,C 180,E1 -11754.414,E2 -11754.414} C_VEL
LIN {X 0,Y 393.056,Z 329.295,A -85,B 0,C 180,E1 -11755.549,E2 -11755.549} C_VEL
LIN {X 0,Y 392.109,Z 338.623,A -85,B 0,C 180,E1 -11756.861,E2 -11756.861} C_VEL
LIN {X 0,Y 391.21,Z 346.919,A -85,B 0,C 180,E1 -11758.3,E2 -11758.3} C_VEL
LIN {X 0,Y 390.375,Z 354.941,A -85,B 0,C 180,E1 -11760.037,E2 -11760.037} C_VEL
LIN {X 0,Y 389.821,Z 360.155,A -85,B 0,C 180,E1 -11761.461,E2 -11761.461} C_VEL
LIN {X 0,Y 389.338,Z 365.105,A -85,B 0,C 180,E1 -11763.174,E2 -11763.174} C_VEL
LIN {X 0,Y 389.044,Z 368.199,A -85,B 0,C 180,E1 -11764.586,E2 -11764.586} C_VEL
LIN {X 0,Y 388.745,Z 371.17,A -85,B 0,C 180,E1 -11766.564,E2 -11766.564} C_VEL
LIN {X 0,Y 388.669,Z 372.192,A -85,B 0,C 180,E1 -11767.683,E2 -11767.683} C_VEL
LIN {X 0,Y 388.607,Z 372.775,A -85,B 0,C 180,E1 -11768.795,E2 -11768.795} C_VEL
LIN {X 0,Y 388.571,Z 372.824,A -85,B 0,C 180,E1 -11770.136,E2 -11770.136} C_VEL
LIN {X 0,Y 388.576,Z 371.767,A -85,B 0,C 180,E1 -11772.093,E2 -11772.093} C_VEL
LIN {X 0,Y 388.717,Z 370.25,A -85,B 0,C 180,E1 -11773.381,E2 -11773.381} C_VEL
LIN {X 0,Y 388.974,Z 366.736,A -85,B 0,C 180,E1 -11775.348,E2 -11775.348} C_VEL
LIN {X 0,Y 389.277,Z 362.072,A -85,B 0,C 180,E1 -11777.136,E2 -11777.136} C_VEL
LIN {X 0,Y 389.662,Z 356.274,A -85,B 0,C 180,E1 -11778.82,E2 -11778.82} C_VEL
LIN {X 0,Y 390.19,Z 349.35,A -85,B 0,C 180,E1 -11780.409,E2 -11780.409} C_VEL
LIN {X 0,Y 390.73,Z 342.287,A -85,B 0,C 180,E1 -11781.727,E2 -11781.727} C_VEL
LIN {X 0,Y 391.439,Z 333.755,A -85,B 0,C 180,E1 -11783.039,E2 -11783.039} C_VEL
LIN {X 0,Y 392.294,Z 323.186,A -85,B 0,C 180,E1 -11784.345,E2 -11784.345} C_VEL
LIN {X 0,Y 393.176,Z 311.266,A -85,B 0,C 180,E1 -11785.515,E2 -11785.515} C_VEL
LIN {X 0,Y 393.893,Z 298.512,A -85,B 0,C 180,E1 -11786.471,E2 -11786.471} C_VEL
LIN {X 0,Y 394.483,Z 285.692,A -85,B 0,C 180,E1 -11787.185,E2 -11787.185} C_VEL
LIN {X 0,Y 394.891,Z 273.616,A -85,B 0,C 180,E1 -11787.652,E2 -11787.652} C_VEL
LIN {X 0,Y 395.191,Z 257.085,A -85,B 0,C 180,E1 -11788.022,E2 -11788.022} C_VEL
LIN {X 0,Y 395.47,Z 235.033,A -85,B 0,C 180,E1 -11788.426,E2 -11788.426} C_VEL
LIN {X 0,Y 395.02,Z 229.217,A -85,B 0,C 180,E1 -11788.555,E2 -11788.555} C_VEL
LIN {X 0,Y 389.8,Z 210.472,A -85,B 0,C 180,E1 -11789.128,E2 -11789.128} C_VEL
LIN {X 0,Y 389.173,Z 204.658,A -85,B 0,C 180,E1 -11789.267,E2 -11789.267} C_VEL
LIN {X 0,Y 389.375,Z 184.42,A -85,B 0,C 180,E1 -11789.649,E2 -11789.649} C_VEL
LIN {X 0,Y 385.111,Z 162.078,A -85,B 0,C 180,E1 -11790.308,E2 -11790.308} C_VEL
LIN {X 0,Y 383.48,Z 151.872,A -85,B 0,C 180,E1 -11792.889,E2 -11792.889} C_VEL
LIN {X 0,Y 383.184,Z 150.759,A -85,B 0,C 180,E1 -11793.22,E2 -11793.22} C_VEL
LIN {X 0,Y 383.228,Z 150.747,A -85,B 0,C 180,E1 -11796.317,E2 -11796.317} C_VEL
LIN {X 0,Y 383.169,Z 150.753,A -85,B 0,C 180,E1 -11798.438,E2 -11798.438} C_VEL
LIN {X 0,Y 383.079,Z 150.768,A -85,B 0,C 180,E1 -11801.643,E2 -11801.643} C_VEL
LIN {X 0,Y 383.048,Z 150.773,A -85,B 0,C 180,E1 -11803.799,E2 -11803.799} C_VEL
LIN {X 0,Y 383.019,Z 150.775,A -85,B 0,C 180,E1 -11807.421,E2 -11807.421} C_VEL
LIN {X 0,Y 383.008,Z 150.772,A -85,B 0,C 180,E1 -11810.64,E2 -11810.64} C_VEL
LIN {X 0,Y 383,Z 150.776,A -85,B 0,C 180,E1 -11813.81,E2 -11813.81} C_VEL
LIN {X 0,Y 382.961,Z 150.784,A -85,B 0,C 180,E1 -11817.31,E2 -11817.31} C_VEL
LIN {X 0,Y 382.974,Z 150.779,A -85,B 0,C 180,E1 -11820.92,E2 -11820.92} C_VEL
LIN {X 0,Y 383.008,Z 150.774,A -85,B 0,C 180,E1 -11824.669,E2 -11824.669} C_VEL
LIN {X 0,Y 382.989,Z 150.775,A -85,B 0,C 180,E1 -11827.903,E2 -11827.903} C_VEL
LIN {X 0,Y 382.958,Z 150.782,A -85,B 0,C 180,E1 -11831.351,E2 -11831.351} C_VEL
LIN {X 0,Y 382.987,Z 150.775,A -85,B 0,C 180,E1 -11834.303,E2 -11834.303} C_VEL
LIN {X 0,Y 382.981,Z 150.779,A -85,B 0,C 180,E1 -11837.237,E2 -11837.237} C_VEL
LIN {X 0,Y 382.984,Z 150.778,A -85,B 0,C 180,E1 -11840.42,E2 -11840.42} C_VEL
LIN {X 0,Y 383.012,Z 150.772,A -85,B 0,C 180,E1 -11844.044,E2 -11844.044} C_VEL
LIN {X 0,Y 382.982,Z 150.775,A -85,B 0,C 180,E1 -11847.58,E2 -11847.58} C_VEL
LIN {X 0,Y 382.974,Z 150.78,A -85,B 0,C 180,E1 -11850.299,E2 -11850.299} C_VEL
LIN {X 0,Y 383.003,Z 150.775,A -85,B 0,C 180,E1 -11854.046,E2 -11854.046} C_VEL
LIN {X 0,Y 382.984,Z 150.775,A -85,B 0,C 180,E1 -11857.334,E2 -11857.334} C_VEL
LIN {X 0,Y 383.011,Z 150.774,A -85,B 0,C 180,E1 -11860.714,E2 -11860.714} C_VEL
LIN {X 0,Y 383.005,Z 150.777,A -85,B 0,C 180,E1 -11864.024,E2 -11864.024} C_VEL
LIN {X 0,Y 383.112,Z 150.759,A -85,B 0,C 180,E1 -11867.284,E2 -11867.284} C_VEL
LIN {X 0,Y 383.139,Z 150.758,A -85,B 0,C 180,E1 -11870.498,E2 -11870.498} C_VEL
LIN {X 0,Y 383.207,Z 150.748,A -85,B 0,C 180,E1 -11872.625,E2 -11872.625} C_VEL
LIN {X 0,Y 383.173,Z 150.752,A -85,B 0,C 180,E1 -11874.739,E2 -11874.739} C_VEL
LIN {X 0,Y 383.372,Z 150.734,A -85,B 0,C 180,E1 -11877.899,E2 -11877.899} C_VEL
LIN {X 0,Y 383.377,Z 150.729,A -85,B 0,C 180,E1 -11882.102,E2 -11882.102} C_VEL
LIN {X 0,Y 383.236,Z 150.745,A -85,B 0,C 180,E1 -11886.318,E2 -11886.318} C_VEL
LIN {X 0,Y 383.144,Z 150.761,A -85,B 0,C 180,E1 -11889.503,E2 -11889.503} C_VEL
LIN {X 0,Y 383.131,Z 150.763,A -85,B 0,C 180,E1 -11893.536,E2 -11893.536} C_VEL
LIN {X 0,Y 383.058,Z 150.772,A -85,B 0,C 180,E1 -11897.435,E2 -11897.435} C_VEL
LIN {X 0,Y 383.022,Z 150.771,A -85,B 0,C 180,E1 -11900.642,E2 -11900.642} C_VEL
LIN {X 0,Y 383.012,Z 150.773,A -85,B 0,C 180,E1 -11903.809,E2 -11903.809} C_VEL
LIN {X 0,Y 382.974,Z 150.781,A -85,B 0,C 180,E1 -11907.309,E2 -11907.309} C_VEL
LIN {X 0,Y 382.984,Z 150.78,A -85,B 0,C 180,E1 -11910.919,E2 -11910.919} C_VEL
LIN {X 0,Y 383.016,Z 150.775,A -85,B 0,C 180,E1 -11914.669,E2 -11914.669} C_VEL
LIN {X 0,Y 382.999,Z 150.773,A -85,B 0,C 180,E1 -11917.903,E2 -11917.903} C_VEL
LIN {X 0,Y 382.965,Z 150.779,A -85,B 0,C 180,E1 -11921.351,E2 -11921.351} C_VEL
LIN {X 0,Y 382.993,Z 150.776,A -85,B 0,C 180,E1 -11924.302,E2 -11924.302} C_VEL
LIN {X 0,Y 383,Z 150.774,A -85,B 0,C 180,E1 -11927.238,E2 -11927.238} C_VEL
LIN {X 0,Y 382.99,Z 150.779,A -85,B 0,C 180,E1 -11930.419,E2 -11930.419} C_VEL
LIN {X 0,Y 383.027,Z 150.772,A -85,B 0,C 180,E1 -11934.044,E2 -11934.044} C_VEL
LIN {X 0,Y 382.989,Z 150.775,A -85,B 0,C 180,E1 -11937.578,E2 -11937.578} C_VEL
LIN {X 0,Y 382.991,Z 150.781,A -85,B 0,C 180,E1 -11940.3,E2 -11940.3} C_VEL
LIN {X 0,Y 383.075,Z 150.899,A -85,B 0,C 180,E1 -11941.553,E2 -11941.553} C_VEL
LIN {X 0,Y 385.979,Z 165.697,A -85,B 0,C 180,E1 -11944.954,E2 -11944.954} C_VEL
LIN {X 0,Y 386.002,Z 170.307,A -85,B 0,C 180,E1 -11945.944,E2 -11945.944} C_VEL
LIN {X 0,Y 384.646,Z 188.326,A -85,B 0,C 180,E1 -11949.715,E2 -11949.715} C_VEL
LIN {X 0,Y 389.053,Z 220.555,A -85,B 0,C 180,E1 -11950.535,E2 -11950.535} C_VEL
LIN {X 0,Y 387.95,Z 297.385,A -85,B 0,C 180,E1 -11951.995,E2 -11951.995} C_VEL
LIN {X 0,Y 387.36,Z 311.197,A -85,B 0,C 180,E1 -11952.478,E2 -11952.478} C_VEL
LIN {X 0,Y 386.606,Z 324.127,A -85,B 0,C 180,E1 -11953.158,E2 -11953.158} C_VEL
LIN {X 0,Y 385.791,Z 335.932,A -85,B 0,C 180,E1 -11954.006,E2 -11954.006} C_VEL
LIN {X 0,Y 384.925,Z 347.324,A -85,B 0,C 180,E1 -11955.054,E2 -11955.054} C_VEL
LIN {X 0,Y 384.166,Z 357.584,A -85,B 0,C 180,E1 -11956.242,E2 -11956.242} C_VEL
LIN {X 0,Y 383.44,Z 366.798,A -85,B 0,C 180,E1 -11957.563,E2 -11957.563} C_VEL
LIN {X 0,Y 382.649,Z 375.763,A -85,B 0,C 180,E1 -11959.149,E2 -11959.149} C_VEL
LIN {X 0,Y 382.158,Z 382.964,A -85,B 0,C 180,E1 -11960.74,E2 -11960.74} C_VEL
LIN {X 0,Y 381.834,Z 389.511,A -85,B 0,C 180,E1 -11962.597,E2 -11962.597} C_VEL
LIN {X 0,Y 381.67,Z 393.165,A -85,B 0,C 180,E1 -11963.908,E2 -11963.908} C_VEL
LIN {X 0,Y 381.63,Z 397.055,A -85,B 0,C 180,E1 -11965.775,E2 -11965.775} C_VEL
LIN {X 0,Y 381.563,Z 398.655,A -85,B 0,C 180,E1 -11966.832,E2 -11966.832} C_VEL
LIN {X 0,Y 381.62,Z 399.847,A -85,B 0,C 180,E1 -11967.889,E2 -11967.889} C_VEL
LIN {X 0,Y 381.674,Z 400.589,A -85,B 0,C 180,E1 -11968.945,E2 -11968.945} C_VEL
LIN {X 0,Y 381.659,Z 400.932,A -85,B 0,C 180,E1 -11970,E2 -11970} C_VEL
LIN {X 0,Y 381.642,Z 400.887,A -85,B 0,C 180,E1 -11971.055,E2 -11971.055} C_VEL
LIN {X 0,Y 381.598,Z 400.451,A -85,B 0,C 180,E1 -11972.111,E2 -11972.111} C_VEL
LIN {X 0,Y 381.624,Z 398.305,A -85,B 0,C 180,E1 -11974.224,E2 -11974.224} C_VEL
LIN {X 0,Y 381.64,Z 395.132,A -85,B 0,C 180,E1 -11976.049,E2 -11976.049} C_VEL
LIN {X 0,Y 381.945,Z 390.472,A -85,B 0,C 180,E1 -11977.932,E2 -11977.932} C_VEL
LIN {X 0,Y 382.449,Z 384.27,A -85,B 0,C 180,E1 -11979.787,E2 -11979.787} C_VEL
LIN {X 0,Y 383.044,Z 377.537,A -85,B 0,C 180,E1 -11981.375,E2 -11981.375} C_VEL
LIN {X 0,Y 384.065,Z 369.21,A -85,B 0,C 180,E1 -11982.954,E2 -11982.954} C_VEL
LIN {X 0,Y 384.955,Z 359.341,A -85,B 0,C 180,E1 -11984.453,E2 -11984.453} C_VEL
LIN {X 0,Y 386.057,Z 349,A -85,B 0,C 180,E1 -11985.711,E2 -11985.711} C_VEL
LIN {X 0,Y 387.152,Z 338.367,A -85,B 0,C 180,E1 -11986.749,E2 -11986.749} C_VEL
LIN {X 0,Y 388.264,Z 326.49,A -85,B 0,C 180,E1 -11987.649,E2 -11987.649} C_VEL
LIN {X 0,Y 389.159,Z 314.185,A -85,B 0,C 180,E1 -11988.355,E2 -11988.355} C_VEL
LIN {X 0,Y 389.953,Z 301.568,A -85,B 0,C 180,E1 -11988.861,E2 -11988.861} C_VEL
LIN {X 0,Y 390.4,Z 287.942,A -85,B 0,C 180,E1 -11989.191,E2 -11989.191} C_VEL
LIN {X 0,Y 391.374,Z 219.379,A -85,B 0,C 180,E1 -11990.498,E2 -11990.498} C_VEL
LIN {X 0,Y 387.685,Z 197.201,A -85,B 0,C 180,E1 -11991.184,E2 -11991.184} C_VEL
LIN {X 0,Y 385.739,Z 187.512,A -85,B 0,C 180,E1 -11991.534,E2 -11991.534} C_VEL
LIN {X 0,Y 387.148,Z 172.234,A -85,B 0,C 180,E1 -11994.815,E2 -11994.815} C_VEL
LIN {X 0,Y 386.739,Z 167.726,A -85,B 0,C 180,E1 -11995.858,E2 -11995.858} C_VEL
LIN {X 0,Y 384.35,Z 156.469,A -85,B 0,C 180,E1 -11998.633,E2 -11998.633} C_VEL
LIN {X 0,Y 383.002,Z 150.779,A -85,B 0,C 180,E1 -12000.112,E2 -12000.112} C_VEL
LIN {X 0,Y 383.002,Z 150.779,A -85,B 0,C 180,E1 -12003.401,E2 -12003.401} C_VEL
LIN {X 0,Y 383.032,Z 150.772,A -85,B 0,C 180,E1 -12006.164,E2 -12006.164} C_VEL
LIN {X 0,Y 382.977,Z 150.776,A -85,B 0,C 180,E1 -12009.962,E2 -12009.962} C_VEL
LIN {X 0,Y 383.008,Z 150.777,A -85,B 0,C 180,E1 -12012.778,E2 -12012.778} C_VEL
LIN {X 0,Y 382.992,Z 150.777,A -85,B 0,C 180,E1 -12015.788,E2 -12015.788} C_VEL
LIN {X 0,Y 382.963,Z 150.781,A -85,B 0,C 180,E1 -12018.8,E2 -12018.8} C_VEL
LIN {X 0,Y 382.993,Z 150.773,A -85,B 0,C 180,E1 -12022.098,E2 -12022.098} C_VEL
LIN {X 0,Y 383.013,Z 150.769,A -85,B 0,C 180,E1 -12025.331,E2 -12025.331} C_VEL
LIN {X 0,Y 382.98,Z 150.773,A -85,B 0,C 180,E1 -12029.081,E2 -12029.081} C_VEL
LIN {X 0,Y 382.967,Z 150.774,A -85,B 0,C 180,E1 -12032.691,E2 -12032.691} C_VEL
LIN {X 0,Y 383.009,Z 150.775,A -85,B 0,C 180,E1 -12036.191,E2 -12036.191} C_VEL
LIN {X 0,Y 383.037,Z 150.77,A -85,B 0,C 180,E1 -12039.597,E2 -12039.597} C_VEL
LIN {X 0,Y 383.042,Z 150.767,A -85,B 0,C 180,E1 -12042.928,E2 -12042.928} C_VEL
LIN {X 0,Y 383.128,Z 150.751,A -85,B 0,C 180,E1 -12046.464,E2 -12046.464} C_VEL
LIN {X 0,Y 383.14,Z 150.754,A -85,B 0,C 180,E1 -12050.497,E2 -12050.497} C_VEL
LIN {X 0,Y 383.242,Z 150.744,A -85,B 0,C 180,E1 -12053.682,E2 -12053.682} C_VEL
LIN {X 0,Y 383.375,Z 150.726,A -85,B 0,C 180,E1 -12057.898,E2 -12057.898} C_VEL
LIN {X 0,Y 383.265,Z 150.737,A -85,B 0,C 180,E1 -12061.05,E2 -12061.05} C_VEL
LIN {X 0,Y 383.238,Z 150.744,A -85,B 0,C 180,E1 -12063.153,E2 -12063.153} C_VEL
LIN {X 0,Y 383.229,Z 150.74,A -85,B 0,C 180,E1 -12066.482,E2 -12066.482} C_VEL
LIN {X 0,Y 383.145,Z 150.754,A -85,B 0,C 180,E1 -12069.502,E2 -12069.502} C_VEL
LIN {X 0,Y 383.138,Z 150.759,A -85,B 0,C 180,E1 -12072.715,E2 -12072.715} C_VEL
LIN {X 0,Y 383.081,Z 150.765,A -85,B 0,C 180,E1 -12075.973,E2 -12075.973} C_VEL
LIN {X 0,Y 383.059,Z 150.77,A -85,B 0,C 180,E1 -12079.283,E2 -12079.283} C_VEL
LIN {X 0,Y 382.991,Z 150.775,A -85,B 0,C 180,E1 -12082.665,E2 -12082.665} C_VEL
LIN {X 0,Y 383.079,Z 150.766,A -85,B 0,C 180,E1 -12086.123,E2 -12086.123} C_VEL
LIN {X 0,Y 382.992,Z 150.778,A -85,B 0,C 180,E1 -12089.699,E2 -12089.699} C_VEL
LIN {X 0,Y 383.002,Z 150.776,A -85,B 0,C 180,E1 -12093.4,E2 -12093.4} C_VEL
LIN {X 0,Y 383.031,Z 150.777,A -85,B 0,C 180,E1 -12096.164,E2 -12096.164} C_VEL
LIN {X 0,Y 383.007,Z 150.779,A -85,B 0,C 180,E1 -12099.958,E2 -12099.958} C_VEL
LIN {X 0,Y 383.003,Z 150.784,A -85,B 0,C 180,E1 -12102.778,E2 -12102.778} C_VEL
LIN {X 0,Y 383.047,Z 150.974,A -85,B 0,C 180,E1 -12105.315,E2 -12105.315} C_VEL
LIN {X 0,Y 385.63,Z 162.738,A -85,B 0,C 180,E1 -12108.525,E2 -12108.525} C_VEL
LIN {X 0,Y 388.839,Z 171.766,A -85,B 0,C 180,E1 -12108.93,E2 -12108.93} C_VEL
LIN {X 0,Y 392.043,Z 186.169,A -85,B 0,C 180,E1 -12109.433,E2 -12109.433} C_VEL
LIN {X 0,Y 390.505,Z 270.015,A -85,B 0,C 180,E1 -12111.04,E2 -12111.04} C_VEL
LIN {X 0,Y 389.962,Z 283.079,A -85,B 0,C 180,E1 -12111.493,E2 -12111.493} C_VEL
LIN {X 0,Y 389.312,Z 295.52,A -85,B 0,C 180,E1 -12112.137,E2 -12112.137} C_VEL
LIN {X 0,Y 388.468,Z 307.067,A -85,B 0,C 180,E1 -12112.94,E2 -12112.94} C_VEL
LIN {X 0,Y 387.353,Z 319.056,A -85,B 0,C 180,E1 -12114.027,E2 -12114.027} C_VEL
LIN {X 0,Y 386.33,Z 329.148,A -85,B 0,C 180,E1 -12115.18,E2 -12115.18} C_VEL
LIN {X 0,Y 385.3,Z 338.568,A -85,B 0,C 180,E1 -12116.511,E2 -12116.511} C_VEL
LIN {X 0,Y 384.351,Z 346.921,A -85,B 0,C 180,E1 -12117.976,E2 -12117.976} C_VEL
LIN {X 0,Y 383.605,Z 353.71,A -85,B 0,C 180,E1 -12119.437,E2 -12119.437} C_VEL
LIN {X 0,Y 382.972,Z 359.26,A -85,B 0,C 180,E1 -12120.902,E2 -12120.902} C_VEL
LIN {X 0,Y 382.388,Z 364.481,A -85,B 0,C 180,E1 -12122.646,E2 -12122.646} C_VEL
LIN {X 0,Y 382.029,Z 368.289,A -85,B 0,C 180,E1 -12124.345,E2 -12124.345} C_VEL
LIN {X 0,Y 381.716,Z 371.045,A -85,B 0,C 180,E1 -12126.105,E2 -12126.105} C_VEL
LIN {X 0,Y 381.62,Z 372.202,A -85,B 0,C 180,E1 -12127.248,E2 -12127.248} C_VEL
LIN {X 0,Y 381.521,Z 372.892,A -85,B 0,C 180,E1 -12128.382,E2 -12128.382} C_VEL
LIN {X 0,Y 381.486,Z 373.104,A -85,B 0,C 180,E1 -12129.975,E2 -12129.975} C_VEL
LIN {X 0,Y 381.479,Z 372.285,A -85,B 0,C 180,E1 -12131.748,E2 -12131.748} C_VEL
LIN {X 0,Y 381.604,Z 370.684,A -85,B 0,C 180,E1 -12133.27,E2 -12133.27} C_VEL
LIN {X 0,Y 381.828,Z 367.667,A -85,B 0,C 180,E1 -12135.067,E2 -12135.067} C_VEL
LIN {X 0,Y 382.111,Z 363.826,A -85,B 0,C 180,E1 -12136.689,E2 -12136.689} C_VEL
LIN {X 0,Y 382.445,Z 358.718,A -85,B 0,C 180,E1 -12138.338,E2 -12138.338} C_VEL
LIN {X 0,Y 382.914,Z 352.349,A -85,B 0,C 180,E1 -12139.959,E2 -12139.959} C_VEL
LIN {X 0,Y 383.584,Z 344.344,A -85,B 0,C 180,E1 -12141.572,E2 -12141.572} C_VEL
LIN {X 0,Y 384.314,Z 336.152,A -85,B 0,C 180,E1 -12142.91,E2 -12142.91} C_VEL
LIN {X 0,Y 385.137,Z 326.164,A -85,B 0,C 180,E1 -12144.24,E2 -12144.24} C_VEL
LIN {X 0,Y 385.938,Z 316.317,A -85,B 0,C 180,E1 -12145.3,E2 -12145.3} C_VEL
LIN {X 0,Y 386.657,Z 305.149,A -85,B 0,C 180,E1 -12146.261,E2 -12146.261} C_VEL
LIN {X 0,Y 387.289,Z 292.252,A -85,B 0,C 180,E1 -12147.113,E2 -12147.113} C_VEL
LIN {X 0,Y 387.841,Z 279.181,A -85,B 0,C 180,E1 -12147.729,E2 -12147.729} C_VEL
LIN {X 0,Y 388.211,Z 266.39,A -85,B 0,C 180,E1 -12148.112,E2 -12148.112} C_VEL
LIN {X 0,Y 389.173,Z 204.658,A -85,B 0,C 180,E1 -12149.267,E2 -12149.267} C_VEL
LIN {X 0,Y 388.51,Z 198.84,A -85,B 0,C 180,E1 -12149.408,E2 -12149.408} C_VEL
LIN {X 0,Y 385.528,Z 189.577,A -85,B 0,C 180,E1 -12149.72,E2 -12149.72} C_VEL
LIN {X 0,Y 381.444,Z 178.516,A -85,B 0,C 180,E1 -12150.124,E2 -12150.124} C_VEL
LIN {X 0,Y 380.551,Z 174.676,A -85,B 0,C 180,E1 -12150.242,E2 -12150.242} C_VEL
LIN {X 0,Y 378.063,Z 162.329,A -85,B 0,C 180,E1 -12150.633,E2 -12150.633} C_VEL
LIN {X 0,Y 376.541,Z 153.364,A -85,B 0,C 180,E1 -12152.942,E2 -12152.942} C_VEL
LIN {X 0,Y 376.119,Z 151.64,A -85,B 0,C 180,E1 -12153.415,E2 -12153.415} C_VEL
LIN {X 0,Y 376.188,Z 151.623,A -85,B 0,C 180,E1 -12156.436,E2 -12156.436} C_VEL
LIN {X 0,Y 376.102,Z 151.637,A -85,B 0,C 180,E1 -12159.682,E2 -12159.682} C_VEL
LIN {X 0,Y 376.036,Z 151.646,A -85,B 0,C 180,E1 -12163.627,E2 -12163.627} C_VEL
LIN {X 0,Y 375.978,Z 151.654,A -85,B 0,C 180,E1 -12167.577,E2 -12167.577} C_VEL
LIN {X 0,Y 375.975,Z 151.649,A -85,B 0,C 180,E1 -12170.833,E2 -12170.833} C_VEL
LIN {X 0,Y 375.928,Z 151.654,A -85,B 0,C 180,E1 -12174.286,E2 -12174.286} C_VEL
LIN {X 0,Y 375.905,Z 151.657,A -85,B 0,C 180,E1 -12176.661,E2 -12176.661} C_VEL
LIN {X 0,Y 375.909,Z 151.66,A -85,B 0,C 180,E1 -12179.085,E2 -12179.085} C_VEL
LIN {X 0,Y 375.949,Z 151.655,A -85,B 0,C 180,E1 -12181.563,E2 -12181.563} C_VEL
LIN {X 0,Y 375.945,Z 151.656,A -85,B 0,C 180,E1 -12185.417,E2 -12185.417} C_VEL
LIN {X 0,Y 375.931,Z 151.654,A -85,B 0,C 180,E1 -12188.263,E2 -12188.263} C_VEL
LIN {X 0,Y 375.911,Z 151.658,A -85,B 0,C 180,E1 -12191.598,E2 -12191.598} C_VEL
LIN {X 0,Y 375.919,Z 151.659,A -85,B 0,C 180,E1 -12194.731,E2 -12194.731} C_VEL
LIN {X 0,Y 375.906,Z 151.657,A -85,B 0,C 180,E1 -12197.697,E2 -12197.697} C_VEL
LIN {X 0,Y 375.933,Z 151.657,A -85,B 0,C 180,E1 -12200.535,E2 -12200.535} C_VEL
LIN {X 0,Y 375.957,Z 151.651,A -85,B 0,C 180,E1 -12203.498,E2 -12203.498} C_VEL
LIN {X 0,Y 375.957,Z 151.651,A -85,B 0,C 180,E1 -12205.889,E2 -12205.889} C_VEL
LIN {X 0,Y 375.959,Z 151.65,A -85,B 0,C 180,E1 -12209.688,E2 -12209.688} C_VEL
LIN {X 0,Y 375.917,Z 151.658,A -85,B 0,C 180,E1 -12212.136,E2 -12212.136} C_VEL
LIN {X 0,Y 375.937,Z 151.659,A -85,B 0,C 180,E1 -12214.535,E2 -12214.535} C_VEL
LIN {X 0,Y 375.97,Z 151.651,A -85,B 0,C 180,E1 -12216.887,E2 -12216.887} C_VEL
LIN {X 0,Y 375.96,Z 151.657,A -85,B 0,C 180,E1 -12220.338,E2 -12220.338} C_VEL
LIN {X 0,Y 375.956,Z 151.652,A -85,B 0,C 180,E1 -12223.716,E2 -12223.716} C_VEL
LIN {X 0,Y 376.079,Z 151.635,A -85,B 0,C 180,E1 -12227.042,E2 -12227.042} C_VEL
LIN {X 0,Y 376.11,Z 151.635,A -85,B 0,C 180,E1 -12230.319,E2 -12230.319} C_VEL
LIN {X 0,Y 376.197,Z 151.623,A -85,B 0,C 180,E1 -12233.565,E2 -12233.565} C_VEL
LIN {X 0,Y 376.336,Z 151.61,A -85,B 0,C 180,E1 -12237.86,E2 -12237.86} C_VEL
LIN {X 0,Y 376.341,Z 151.605,A -85,B 0,C 180,E1 -12242.141,E2 -12242.141} C_VEL
LIN {X 0,Y 376.196,Z 151.621,A -85,B 0,C 180,E1 -12246.436,E2 -12246.436} C_VEL
LIN {X 0,Y 376.115,Z 151.637,A -85,B 0,C 180,E1 -12249.682,E2 -12249.682} C_VEL
LIN {X 0,Y 376.095,Z 151.638,A -85,B 0,C 180,E1 -12253.658,E2 -12253.658} C_VEL
LIN {X 0,Y 376.012,Z 151.648,A -85,B 0,C 180,E1 -12257.59,E2 -12257.59} C_VEL
LIN {X 0,Y 375.984,Z 151.649,A -85,B 0,C 180,E1 -12260.832,E2 -12260.832} C_VEL
LIN {X 0,Y 375.972,Z 151.649,A -85,B 0,C 180,E1 -12264.284,E2 -12264.284} C_VEL
LIN {X 0,Y 375.922,Z 151.655,A -85,B 0,C 180,E1 -12267.865,E2 -12267.865} C_VEL
LIN {X 0,Y 375.942,Z 151.655,A -85,B 0,C 180,E1 -12270.689,E2 -12270.689} C_VEL
LIN {X 0,Y 375.962,Z 151.65,A -85,B 0,C 180,E1 -12274.112,E2 -12274.112} C_VEL
LIN {X 0,Y 375.954,Z 151.656,A -85,B 0,C 180,E1 -12276.742,E2 -12276.742} C_VEL
LIN {X 0,Y 375.943,Z 151.652,A -85,B 0,C 180,E1 -12279.962,E2 -12279.962} C_VEL
LIN {X 0,Y 375.929,Z 151.654,A -85,B 0,C 180,E1 -12283.767,E2 -12283.767} C_VEL
LIN {X 0,Y 375.937,Z 151.658,A -85,B 0,C 180,E1 -12286.811,E2 -12286.811} C_VEL
LIN {X 0,Y 375.939,Z 151.659,A -85,B 0,C 180,E1 -12290.534,E2 -12290.534} C_VEL
LIN {X 0,Y 375.966,Z 151.649,A -85,B 0,C 180,E1 -12293.496,E2 -12293.496} C_VEL
LIN {X 0,Y 375.963,Z 151.651,A -85,B 0,C 180,E1 -12295.888,E2 -12295.888} C_VEL
LIN {X 0,Y 375.966,Z 151.654,A -85,B 0,C 180,E1 -12299.687,E2 -12299.687} C_VEL
LIN {X 0,Y 376.026,Z 151.83,A -85,B 0,C 180,E1 -12301.323,E2 -12301.323} C_VEL
LIN {X 0,Y 378.906,Z 166.434,A -85,B 0,C 180,E1 -12304.747,E2 -12304.747} C_VEL
LIN {X 0,Y 379.131,Z 170.253,A -85,B 0,C 180,E1 -12305.595,E2 -12305.595} C_VEL
LIN {X 0,Y 377.683,Z 188.082,A -85,B 0,C 180,E1 -12309.389,E2 -12309.389} C_VEL
LIN {X 0,Y 382.23,Z 220.956,A -85,B 0,C 180,E1 -12310.249,E2 -12310.249} C_VEL
LIN {X 0,Y 381.09,Z 297.32,A -85,B 0,C 180,E1 -12311.729,E2 -12311.729} C_VEL
LIN {X 0,Y 380.494,Z 311.07,A -85,B 0,C 180,E1 -12312.221,E2 -12312.221} C_VEL
LIN {X 0,Y 379.679,Z 323.948,A -85,B 0,C 180,E1 -12312.911,E2 -12312.911} C_VEL
LIN {X 0,Y 378.799,Z 336.537,A -85,B 0,C 180,E1 -12313.841,E2 -12313.841} C_VEL
LIN {X 0,Y 377.917,Z 347.769,A -85,B 0,C 180,E1 -12314.909,E2 -12314.909} C_VEL
LIN {X 0,Y 377.23,Z 356.862,A -85,B 0,C 180,E1 -12315.983,E2 -12315.983} C_VEL
LIN {X 0,Y 376.456,Z 366.173,A -85,B 0,C 180,E1 -12317.328,E2 -12317.328} C_VEL
LIN {X 0,Y 375.628,Z 375.209,A -85,B 0,C 180,E1 -12318.943,E2 -12318.943} C_VEL
LIN {X 0,Y 375.113,Z 382.48,A -85,B 0,C 180,E1 -12320.564,E2 -12320.564} C_VEL
LIN {X 0,Y 374.844,Z 387.38,A -85,B 0,C 180,E1 -12321.916,E2 -12321.916} C_VEL
LIN {X 0,Y 374.625,Z 392.127,A -85,B 0,C 180,E1 -12323.537,E2 -12323.537} C_VEL
LIN {X 0,Y 374.551,Z 395.742,A -85,B 0,C 180,E1 -12325.156,E2 -12325.156} C_VEL
LIN {X 0,Y 374.477,Z 398.325,A -85,B 0,C 180,E1 -12326.772,E2 -12326.772} C_VEL
LIN {X 0,Y 374.52,Z 399.538,A -85,B 0,C 180,E1 -12327.849,E2 -12327.849} C_VEL
LIN {X 0,Y 374.588,Z 400.306,A -85,B 0,C 180,E1 -12328.925,E2 -12328.925} C_VEL
LIN {X 0,Y 374.591,Z 400.665,A -85,B 0,C 180,E1 -12330,E2 -12330} C_VEL
LIN {X 0,Y 374.557,Z 400.635,A -85,B 0,C 180,E1 -12331.075,E2 -12331.075} C_VEL
LIN {X 0,Y 374.497,Z 400.217,A -85,B 0,C 180,E1 -12332.151,E2 -12332.151} C_VEL
LIN {X 0,Y 374.463,Z 399.375,A -85,B 0,C 180,E1 -12333.228,E2 -12333.228} C_VEL
LIN {X 0,Y 374.527,Z 398.119,A -85,B 0,C 180,E1 -12334.305,E2 -12334.305} C_VEL
LIN {X 0,Y 374.546,Z 395.291,A -85,B 0,C 180,E1 -12336.011,E2 -12336.011} C_VEL
LIN {X 0,Y 374.888,Z 390.371,A -85,B 0,C 180,E1 -12338.083,E2 -12338.083} C_VEL
LIN {X 0,Y 375.416,Z 384.227,A -85,B 0,C 180,E1 -12339.972,E2 -12339.972} C_VEL
LIN {X 0,Y 376.076,Z 377.542,A -85,B 0,C 180,E1 -12341.589,E2 -12341.589} C_VEL
LIN {X 0,Y 377.122,Z 369.271,A -85,B 0,C 180,E1 -12343.196,E2 -12343.196} C_VEL
LIN {X 0,Y 378.01,Z 360.127,A -85,B 0,C 180,E1 -12344.636,E2 -12344.636} C_VEL
LIN {X 0,Y 379.227,Z 349.245,A -85,B 0,C 180,E1 -12346.002,E2 -12346.002} C_VEL
LIN {X 0,Y 380.367,Z 338.728,A -85,B 0,C 180,E1 -12347.057,E2 -12347.057} C_VEL
LIN {X 0,Y 381.547,Z 327.083,A -85,B 0,C 180,E1 -12347.971,E2 -12347.971} C_VEL
LIN {X 0,Y 382.572,Z 313.751,A -85,B 0,C 180,E1 -12348.753,E2 -12348.753} C_VEL
LIN {X 0,Y 383.398,Z 301.05,A -85,B 0,C 180,E1 -12349.266,E2 -12349.266} C_VEL
LIN {X 0,Y 383.859,Z 286.922,A -85,B 0,C 180,E1 -12349.607,E2 -12349.607} C_VEL
LIN {X 0,Y 384.895,Z 220.447,A -85,B 0,C 180,E1 -12350.894,E2 -12350.894} C_VEL
LIN {X 0,Y 381.416,Z 199.271,A -85,B 0,C 180,E1 -12351.566,E2 -12351.566} C_VEL
LIN {X 0,Y 378.977,Z 187.174,A -85,B 0,C 180,E1 -12352.027,E2 -12352.027} C_VEL
LIN {X 0,Y 380.304,Z 172.929,A -85,B 0,C 180,E1 -12355.153,E2 -12355.153} C_VEL
LIN {X 0,Y 379.163,Z 165.744,A -85,B 0,C 180,E1 -12356.897,E2 -12356.897} C_VEL
LIN {X 0,Y 376.482,Z 153.821,A -85,B 0,C 180,E1 -12359.958,E2 -12359.958} C_VEL
LIN {X 0,Y 375.956,Z 151.659,A -85,B 0,C 180,E1 -12360.591,E2 -12360.591} C_VEL
LIN {X 0,Y 375.961,Z 151.649,A -85,B 0,C 180,E1 -12364.111,E2 -12364.111} C_VEL
LIN {X 0,Y 375.954,Z 151.651,A -85,B 0,C 180,E1 -12366.741,E2 -12366.741} C_VEL
LIN {X 0,Y 375.94,Z 151.653,A -85,B 0,C 180,E1 -12369.961,E2 -12369.961} C_VEL
LIN {X 0,Y 375.927,Z 151.655,A -85,B 0,C 180,E1 -12373.766,E2 -12373.766} C_VEL
LIN {X 0,Y 375.934,Z 151.656,A -85,B 0,C 180,E1 -12376.811,E2 -12376.811} C_VEL
LIN {X 0,Y 375.936,Z 151.657,A -85,B 0,C 180,E1 -12380.533,E2 -12380.533} C_VEL
LIN {X 0,Y 375.958,Z 151.653,A -85,B 0,C 180,E1 -12383.497,E2 -12383.497} C_VEL
LIN {X 0,Y 375.959,Z 151.647,A -85,B 0,C 180,E1 -12385.888,E2 -12385.888} C_VEL
LIN {X 0,Y 375.961,Z 151.646,A -85,B 0,C 180,E1 -12389.686,E2 -12389.686} C_VEL
LIN {X 0,Y 375.918,Z 151.658,A -85,B 0,C 180,E1 -12392.134,E2 -12392.134} C_VEL
LIN {X 0,Y 375.938,Z 151.654,A -85,B 0,C 180,E1 -12394.533,E2 -12394.533} C_VEL
LIN {X 0,Y 375.971,Z 151.643,A -85,B 0,C 180,E1 -12396.886,E2 -12396.886} C_VEL
LIN {X 0,Y 375.961,Z 151.653,A -85,B 0,C 180,E1 -12400.337,E2 -12400.337} C_VEL
LIN {X 0,Y 375.963,Z 151.65,A -85,B 0,C 180,E1 -12403.715,E2 -12403.715} C_VEL
LIN {X 0,Y 376.105,Z 151.624,A -85,B 0,C 180,E1 -12407.042,E2 -12407.042} C_VEL
LIN {X 0,Y 376.111,Z 151.631,A -85,B 0,C 180,E1 -12410.318,E2 -12410.318} C_VEL
LIN {X 0,Y 376.201,Z 151.62,A -85,B 0,C 180,E1 -12413.564,E2 -12413.564} C_VEL
LIN {X 0,Y 376.34,Z 151.602,A -85,B 0,C 180,E1 -12417.859,E2 -12417.859} C_VEL
LIN {X 0,Y 376.236,Z 151.612,A -85,B 0,C 180,E1 -12421.07,E2 -12421.07} C_VEL
LIN {X 0,Y 376.351,Z 151.6,A -85,B 0,C 180,E1 -12422.14,E2 -12422.14} C_VEL
LIN {X 0,Y 376.199,Z 151.616,A -85,B 0,C 180,E1 -12426.466,E2 -12426.466} C_VEL
LIN {X 0,Y 376.115,Z 151.628,A -85,B 0,C 180,E1 -12429.681,E2 -12429.681} C_VEL
LIN {X 0,Y 376.091,Z 151.633,A -85,B 0,C 180,E1 -12433.657,E2 -12433.657} C_VEL
LIN {X 0,Y 376.033,Z 151.642,A -85,B 0,C 180,E1 -12437.399,E2 -12437.399} C_VEL
LIN {X 0,Y 375.979,Z 151.653,A -85,B 0,C 180,E1 -12440.831,E2 -12440.831} C_VEL
LIN {X 0,Y 375.987,Z 151.652,A -85,B 0,C 180,E1 -12444.281,E2 -12444.281} C_VEL
LIN {X 0,Y 376.019,Z 151.65,A -85,B 0,C 180,E1 -12446.651,E2 -12446.651} C_VEL
LIN {X 0,Y 375.97,Z 151.655,A -85,B 0,C 180,E1 -12449.078,E2 -12449.078} C_VEL
LIN {X 0,Y 375.948,Z 151.655,A -85,B 0,C 180,E1 -12452.828,E2 -12452.828} C_VEL
LIN {X 0,Y 375.956,Z 151.655,A -85,B 0,C 180,E1 -12455.415,E2 -12455.415} C_VEL
LIN {X 0,Y 375.972,Z 151.654,A -85,B 0,C 180,E1 -12458.27,E2 -12458.27} C_VEL
LIN {X 0,Y 375.932,Z 151.66,A -85,B 0,C 180,E1 -12461.6,E2 -12461.6} C_VEL
LIN {X 0,Y 375.964,Z 151.677,A -85,B 0,C 180,E1 -12464.847,E2 -12464.847} C_VEL
LIN {X 0,Y 378.495,Z 163.058,A -85,B 0,C 180,E1 -12468.013,E2 -12468.013} C_VEL
LIN {X 0,Y 382.51,Z 173.614,A -85,B 0,C 180,E1 -12468.528,E2 -12468.528} C_VEL
LIN {X 0,Y 385.593,Z 187.539,A -85,B 0,C 180,E1 -12469.034,E2 -12469.034} C_VEL
LIN {X 0,Y 383.953,Z 270.459,A -85,B 0,C 180,E1 -12470.649,E2 -12470.649} C_VEL
LIN {X 0,Y 383.381,Z 283.452,A -85,B 0,C 180,E1 -12471.108,E2 -12471.108} C_VEL
LIN {X 0,Y 382.669,Z 296.187,A -85,B 0,C 180,E1 -12471.78,E2 -12471.78} C_VEL
LIN {X 0,Y 381.802,Z 307.589,A -85,B 0,C 180,E1 -12472.595,E2 -12472.595} C_VEL
LIN {X 0,Y 380.694,Z 318.821,A -85,B 0,C 180,E1 -12473.625,E2 -12473.625} C_VEL
LIN {X 0,Y 379.637,Z 329.034,A -85,B 0,C 180,E1 -12474.803,E2 -12474.803} C_VEL
LIN {X 0,Y 378.529,Z 338.512,A -85,B 0,C 180,E1 -12476.151,E2 -12476.151} C_VEL
LIN {X 0,Y 377.524,Z 346.927,A -85,B 0,C 180,E1 -12477.642,E2 -12477.642} C_VEL
LIN {X 0,Y 376.549,Z 354.956,A -85,B 0,C 180,E1 -12479.419,E2 -12479.419} C_VEL
LIN {X 0,Y 375.92,Z 360.337,A -85,B 0,C 180,E1 -12480.917,E2 -12480.917} C_VEL
LIN {X 0,Y 375.304,Z 365.376,A -85,B 0,C 180,E1 -12482.691,E2 -12482.691} C_VEL
LIN {X 0,Y 374.916,Z 369.076,A -85,B 0,C 180,E1 -12484.46,E2 -12484.46} C_VEL
LIN {X 0,Y 374.696,Z 370.856,A -85,B 0,C 180,E1 -12485.629,E2 -12485.629} C_VEL
LIN {X 0,Y 374.562,Z 372.221,A -85,B 0,C 180,E1 -12486.837,E2 -12486.837} C_VEL
LIN {X 0,Y 374.454,Z 373.01,A -85,B 0,C 180,E1 -12487.953,E2 -12487.953} C_VEL
LIN {X 0,Y 374.394,Z 373.382,A -85,B 0,C 180,E1 -12489.813,E2 -12489.813} C_VEL
LIN {X 0,Y 374.367,Z 372.796,A -85,B 0,C 180,E1 -12491.389,E2 -12491.389} C_VEL
LIN {X 0,Y 374.495,Z 371.104,A -85,B 0,C 180,E1 -12493.153,E2 -12493.153} C_VEL
LIN {X 0,Y 374.795,Z 367.461,A -85,B 0,C 180,E1 -12495.336,E2 -12495.336} C_VEL
LIN {X 0,Y 375.095,Z 363.415,A -85,B 0,C 180,E1 -12497.007,E2 -12497.007} C_VEL
LIN {X 0,Y 375.547,Z 357.162,A -85,B 0,C 180,E1 -12498.941,E2 -12498.941} C_VEL
LIN {X 0,Y 376.089,Z 350.316,A -85,B 0,C 180,E1 -12500.589,E2 -12500.589} C_VEL
LIN {X 0,Y 376.755,Z 342.655,A -85,B 0,C 180,E1 -12502.078,E2 -12502.078} C_VEL
LIN {X 0,Y 377.425,Z 334.901,A -85,B 0,C 180,E1 -12503.317,E2 -12503.317} C_VEL
LIN {X 0,Y 378.243,Z 325.68,A -85,B 0,C 180,E1 -12504.536,E2 -12504.536} C_VEL
LIN {X 0,Y 379.058,Z 315.636,A -85,B 0,C 180,E1 -12505.614,E2 -12505.614} C_VEL
LIN {X 0,Y 379.817,Z 304.717,A -85,B 0,C 180,E1 -12506.552,E2 -12506.552} C_VEL
LIN {X 0,Y 380.449,Z 291.902,A -85,B 0,C 180,E1 -12507.404,E2 -12507.404} C_VEL
LIN {X 0,Y 380.961,Z 279.734,A -85,B 0,C 180,E1 -12507.985,E2 -12507.985} C_VEL
LIN {X 0,Y 381.381,Z 266.684,A -85,B 0,C 180,E1 -12508.383,E2 -12508.383} C_VEL
LIN {X 0,Y 382.512,Z 185.036,A -85,B 0,C 180,E1 -12509.946,E2 -12509.946} C_VEL
LIN {X 0,Y 380.551,Z 174.676,A -85,B 0,C 180,E1 -12510.242,E2 -12510.242} C_VEL
LIN {X 0,Y 379.161,Z 170.914,A -85,B 0,C 180,E1 -12510.386,E2 -12510.386} C_VEL
LIN {X 0,Y 376.895,Z 167.664,A -85,B 0,C 180,E1 -12510.591,E2 -12510.591} C_VEL
LIN {X 0,Y 373.557,Z 163.954,A -85,B 0,C 180,E1 -12510.97,E2 -12510.97} C_VEL
LIN {X 0,Y 371.192,Z 161.075,A -85,B 0,C 180,E1 -12511.436,E2 -12511.436} C_VEL
LIN {X 0,Y 370.402,Z 159.211,A -85,B 0,C 180,E1 -12511.852,E2 -12511.852} C_VEL
LIN {X 0,Y 369.033,Z 152.525,A -85,B 0,C 180,E1 -12513.651,E2 -12513.651} C_VEL
LIN {X 0,Y 369.15,Z 152.499,A -85,B 0,C 180,E1 -12516.559,E2 -12516.559} C_VEL
LIN {X 0,Y 369.053,Z 152.517,A -85,B 0,C 180,E1 -12519.869,E2 -12519.869} C_VEL
LIN {X 0,Y 368.997,Z 152.524,A -85,B 0,C 180,E1 -12523.749,E2 -12523.749} C_VEL
LIN {X 0,Y 368.932,Z 152.531,A -85,B 0,C 180,E1 -12527.746,E2 -12527.746} C_VEL
LIN {X 0,Y 368.898,Z 152.533,A -85,B 0,C 180,E1 -12531.222,E2 -12531.222} C_VEL
LIN {X 0,Y 368.901,Z 152.532,A -85,B 0,C 180,E1 -12533.873,E2 -12533.873} C_VEL
LIN {X 0,Y 368.852,Z 152.54,A -85,B 0,C 180,E1 -12537.213,E2 -12537.213} C_VEL
LIN {X 0,Y 368.888,Z 152.534,A -85,B 0,C 180,E1 -12539.693,E2 -12539.693} C_VEL
LIN {X 0,Y 368.892,Z 152.535,A -85,B 0,C 180,E1 -12543.043,E2 -12543.043} C_VEL
LIN {X 0,Y 368.908,Z 152.529,A -85,B 0,C 180,E1 -12546.198,E2 -12546.198} C_VEL
LIN {X 0,Y 368.871,Z 152.538,A -85,B 0,C 180,E1 -12548.958,E2 -12548.958} C_VEL
LIN {X 0,Y 368.856,Z 152.535,A -85,B 0,C 180,E1 -12552.006,E2 -12552.006} C_VEL
LIN {X 0,Y 368.872,Z 152.537,A -85,B 0,C 180,E1 -12555.176,E2 -12555.176} C_VEL
LIN {X 0,Y 368.859,Z 152.535,A -85,B 0,C 180,E1 -12558.175,E2 -12558.175} C_VEL
LIN {X 0,Y 368.875,Z 152.534,A -85,B 0,C 180,E1 -12561.367,E2 -12561.367} C_VEL
LIN {X 0,Y 368.93,Z 152.528,A -85,B 0,C 180,E1 -12565.147,E2 -12565.147} C_VEL
LIN {X 0,Y 368.896,Z 152.532,A -85,B 0,C 180,E1 -12569.044,E2 -12569.044} C_VEL
LIN {X 0,Y 368.907,Z 152.529,A -85,B 0,C 180,E1 -12571.559,E2 -12571.559} C_VEL
LIN {X 0,Y 368.92,Z 152.529,A -85,B 0,C 180,E1 -12574.014,E2 -12574.014} C_VEL
LIN {X 0,Y 368.896,Z 152.531,A -85,B 0,C 180,E1 -12577.603,E2 -12577.603} C_VEL
LIN {X 0,Y 368.899,Z 152.53,A -85,B 0,C 180,E1 -12581.103,E2 -12581.103} C_VEL
LIN {X 0,Y 368.923,Z 152.53,A -85,B 0,C 180,E1 -12584.533,E2 -12584.533} C_VEL
LIN {X 0,Y 369.026,Z 152.515,A -85,B 0,C 180,E1 -12586.79,E2 -12586.79} C_VEL
LIN {X 0,Y 369.06,Z 152.516,A -85,B 0,C 180,E1 -12590.132,E2 -12590.132} C_VEL
LIN {X 0,Y 369.16,Z 152.499,A -85,B 0,C 180,E1 -12593.442,E2 -12593.442} C_VEL
LIN {X 0,Y 369.299,Z 152.486,A -85,B 0,C 180,E1 -12597.819,E2 -12597.819} C_VEL
LIN {X 0,Y 369.305,Z 152.482,A -85,B 0,C 180,E1 -12602.182,E2 -12602.182} C_VEL
LIN {X 0,Y 369.158,Z 152.498,A -85,B 0,C 180,E1 -12606.56,E2 -12606.56} C_VEL
LIN {X 0,Y 369.065,Z 152.513,A -85,B 0,C 180,E1 -12609.869,E2 -12609.869} C_VEL
LIN {X 0,Y 369.043,Z 152.515,A -85,B 0,C 180,E1 -12613.773,E2 -12613.773} C_VEL
LIN {X 0,Y 368.958,Z 152.525,A -85,B 0,C 180,E1 -12617.745,E2 -12617.745} C_VEL
LIN {X 0,Y 368.914,Z 152.534,A -85,B 0,C 180,E1 -12621.221,E2 -12621.221} C_VEL
LIN {X 0,Y 368.927,Z 152.528,A -85,B 0,C 180,E1 -12624.778,E2 -12624.778} C_VEL
LIN {X 0,Y 368.897,Z 152.533,A -85,B 0,C 180,E1 -12628.792,E2 -12628.792} C_VEL
LIN {X 0,Y 368.894,Z 152.531,A -85,B 0,C 180,E1 -12632.239,E2 -12632.239} C_VEL
LIN {X 0,Y 368.928,Z 152.532,A -85,B 0,C 180,E1 -12635,E2 -12635} C_VEL
LIN {X 0,Y 368.882,Z 152.536,A -85,B 0,C 180,E1 -12638.634,E2 -12638.634} C_VEL
LIN {X 0,Y 368.874,Z 152.533,A -85,B 0,C 180,E1 -12642.007,E2 -12642.007} C_VEL
LIN {X 0,Y 368.878,Z 152.534,A -85,B 0,C 180,E1 -12645.175,E2 -12645.175} C_VEL
LIN {X 0,Y 368.868,Z 152.536,A -85,B 0,C 180,E1 -12648.175,E2 -12648.175} C_VEL
LIN {X 0,Y 368.881,Z 152.532,A -85,B 0,C 180,E1 -12651.366,E2 -12651.366} C_VEL
LIN {X 0,Y 368.939,Z 152.525,A -85,B 0,C 180,E1 -12655.146,E2 -12655.146} C_VEL
LIN {X 0,Y 368.916,Z 152.532,A -85,B 0,C 180,E1 -12659.045,E2 -12659.045} C_VEL
LIN {X 0,Y 368.949,Z 152.631,A -85,B 0,C 180,E1 -12661.054,E2 -12661.054} C_VEL
LIN {X 0,Y 371.755,Z 166.835,A -85,B 0,C 180,E1 -12664.453,E2 -12664.453} C_VEL
LIN {X 0,Y 372.18,Z 169.236,A -85,B 0,C 180,E1 -12665.013,E2 -12665.013} C_VEL
LIN {X 0,Y 371.323,Z 180.461,A -85,B 0,C 180,E1 -12667.463,E2 -12667.463} C_VEL
LIN {X 0,Y 370.755,Z 187.817,A -85,B 0,C 180,E1 -12669.055,E2 -12669.055} C_VEL
LIN {X 0,Y 375.429,Z 220.894,A -85,B 0,C 180,E1 -12669.945,E2 -12669.945} C_VEL
LIN {X 0,Y 374.29,Z 296.119,A -85,B 0,C 180,E1 -12671.42,E2 -12671.42} C_VEL
LIN {X 0,Y 373.69,Z 309.41,A -85,B 0,C 180,E1 -12671.886,E2 -12671.886} C_VEL
LIN {X 0,Y 372.862,Z 322.746,A -85,B 0,C 180,E1 -12672.589,E2 -12672.589} C_VEL
LIN {X 0,Y 372.082,Z 333.956,A -85,B 0,C 180,E1 -12673.4,E2 -12673.4} C_VEL
LIN {X 0,Y 371.075,Z 345.607,A -85,B 0,C 180,E1 -12674.483,E2 -12674.483} C_VEL
LIN {X 0,Y 370.271,Z 356.114,A -85,B 0,C 180,E1 -12675.714,E2 -12675.714} C_VEL
LIN {X 0,Y 369.449,Z 365.536,A -85,B 0,C 180,E1 -12677.084,E2 -12677.084} C_VEL
LIN {X 0,Y 368.595,Z 374.636,A -85,B 0,C 180,E1 -12678.729,E2 -12678.729} C_VEL
LIN {X 0,Y 368.077,Z 381.968,A -85,B 0,C 180,E1 -12680.382,E2 -12680.382} C_VEL
LIN {X 0,Y 367.781,Z 386.913,A -85,B 0,C 180,E1 -12681.76,E2 -12681.76} C_VEL
LIN {X 0,Y 367.556,Z 391.706,A -85,B 0,C 180,E1 -12683.412,E2 -12683.412} C_VEL
LIN {X 0,Y 367.47,Z 395.362,A -85,B 0,C 180,E1 -12685.063,E2 -12685.063} C_VEL
LIN {X 0,Y 367.394,Z 397.984,A -85,B 0,C 180,E1 -12686.71,E2 -12686.71} C_VEL
LIN {X 0,Y 367.42,Z 399.215,A -85,B 0,C 180,E1 -12687.807,E2 -12687.807} C_VEL
LIN {X 0,Y 367.489,Z 400.018,A -85,B 0,C 180,E1 -12688.904,E2 -12688.904} C_VEL
LIN {X 0,Y 367.507,Z 400.396,A -85,B 0,C 180,E1 -12690,E2 -12690} C_VEL
LIN {X 0,Y 367.459,Z 400.383,A -85,B 0,C 180,E1 -12691.096,E2 -12691.096} C_VEL
LIN {X 0,Y 367.396,Z 399.982,A -85,B 0,C 180,E1 -12692.192,E2 -12692.192} C_VEL
LIN {X 0,Y 367.38,Z 399.176,A -85,B 0,C 180,E1 -12693.29,E2 -12693.29} C_VEL
LIN {X 0,Y 367.434,Z 397.938,A -85,B 0,C 180,E1 -12694.388,E2 -12694.388} C_VEL
LIN {X 0,Y 367.467,Z 395.412,A -85,B 0,C 180,E1 -12695.992,E2 -12695.992} C_VEL
LIN {X 0,Y 367.702,Z 391.705,A -85,B 0,C 180,E1 -12697.689,E2 -12697.689} C_VEL
LIN {X 0,Y 368.132,Z 386.992,A -85,B 0,C 180,E1 -12699.339,E2 -12699.339} C_VEL
LIN {X 0,Y 368.81,Z 379.923,A -85,B 0,C 180,E1 -12701.263,E2 -12701.263} C_VEL
LIN {X 0,Y 369.841,Z 372.293,A -85,B 0,C 180,E1 -12702.902,E2 -12702.902} C_VEL
LIN {X 0,Y 370.942,Z 362.735,A -85,B 0,C 180,E1 -12704.539,E2 -12704.539} C_VEL
LIN {X 0,Y 372.026,Z 352.901,A -85,B 0,C 180,E1 -12705.898,E2 -12705.898} C_VEL
LIN {X 0,Y 373.31,Z 341.92,A -85,B 0,C 180,E1 -12707.107,E2 -12707.107} C_VEL
LIN {X 0,Y 374.465,Z 331.189,A -85,B 0,C 180,E1 -12708.039,E2 -12708.039} C_VEL
LIN {X 0,Y 375.595,Z 318.3,A -85,B 0,C 180,E1 -12708.902,E2 -12708.902} C_VEL
LIN {X 0,Y 376.534,Z 306.009,A -85,B 0,C 180,E1 -12709.49,E2 -12709.49} C_VEL
LIN {X 0,Y 377.178,Z 293.617,A -85,B 0,C 180,E1 -12709.876,E2 -12709.876} C_VEL
LIN {X 0,Y 378.394,Z 221.038,A -85,B 0,C 180,E1 -12711.323,E2 -12711.323} C_VEL
LIN {X 0,Y 374.731,Z 199.01,A -85,B 0,C 180,E1 -12712.052,E2 -12712.052} C_VEL
LIN {X 0,Y 372.215,Z 186.987,A -85,B 0,C 180,E1 -12712.509,E2 -12712.509} C_VEL
LIN {X 0,Y 373.452,Z 174.069,A -85,B 0,C 180,E1 -12715.402,E2 -12715.402} C_VEL
LIN {X 0,Y 371.778,Z 164.886,A -85,B 0,C 180,E1 -12717.704,E2 -12717.704} C_VEL
LIN {X 0,Y 369.255,Z 153.988,A -85,B 0,C 180,E1 -12720.606,E2 -12720.606} C_VEL
LIN {X 0,Y 368.924,Z 152.538,A -85,B 0,C 180,E1 -12721.025,E2 -12721.025} C_VEL
LIN {X 0,Y 368.93,Z 152.525,A -85,B 0,C 180,E1 -12725.001,E2 -12725.001} C_VEL
LIN {X 0,Y 368.879,Z 152.537,A -85,B 0,C 180,E1 -12728.634,E2 -12728.634} C_VEL
LIN {X 0,Y 368.866,Z 152.537,A -85,B 0,C 180,E1 -12732.006,E2 -12732.006} C_VEL
LIN {X 0,Y 368.876,Z 152.54,A -85,B 0,C 180,E1 -12735.175,E2 -12735.175} C_VEL
LIN {X 0,Y 368.862,Z 152.537,A -85,B 0,C 180,E1 -12738.174,E2 -12738.174} C_VEL
LIN {X 0,Y 368.877,Z 152.533,A -85,B 0,C 180,E1 -12741.366,E2 -12741.366} C_VEL
LIN {X 0,Y 368.932,Z 152.523,A -85,B 0,C 180,E1 -12745.145,E2 -12745.145} C_VEL
LIN {X 0,Y 368.898,Z 152.526,A -85,B 0,C 180,E1 -12749.043,E2 -12749.043} C_VEL
LIN {X 0,Y 368.909,Z 152.529,A -85,B 0,C 180,E1 -12751.557,E2 -12751.557} C_VEL
LIN {X 0,Y 368.888,Z 152.532,A -85,B 0,C 180,E1 -12755.219,E2 -12755.219} C_VEL
LIN {X 0,Y 368.886,Z 152.523,A -85,B 0,C 180,E1 -12757.601,E2 -12757.601} C_VEL
LIN {X 0,Y 368.9,Z 152.527,A -85,B 0,C 180,E1 -12761.102,E2 -12761.102} C_VEL
LIN {X 0,Y 368.937,Z 152.529,A -85,B 0,C 180,E1 -12764.532,E2 -12764.532} C_VEL
LIN {X 0,Y 369.06,Z 152.501,A -85,B 0,C 180,E1 -12766.79,E2 -12766.79} C_VEL
LIN {X 0,Y 369.061,Z 152.511,A -85,B 0,C 180,E1 -12770.131,E2 -12770.131} C_VEL
LIN {X 0,Y 369.161,Z 152.496,A -85,B 0,C 180,E1 -12773.44,E2 -12773.44} C_VEL
LIN {X 0,Y 369.304,Z 152.477,A -85,B 0,C 180,E1 -12777.818,E2 -12777.818} C_VEL
LIN {X 0,Y 369.207,Z 152.487,A -85,B 0,C 180,E1 -12781.09,E2 -12781.09} C_VEL
LIN {X 0,Y 369.315,Z 152.477,A -85,B 0,C 180,E1 -12782.181,E2 -12782.181} C_VEL
LIN {X 0,Y 369.163,Z 152.492,A -85,B 0,C 180,E1 -12786.558,E2 -12786.558} C_VEL
LIN {X 0,Y 369.065,Z 152.504,A -85,B 0,C 180,E1 -12789.868,E2 -12789.868} C_VEL
LIN {X 0,Y 369.038,Z 152.51,A -85,B 0,C 180,E1 -12793.772,E2 -12793.772} C_VEL
LIN {X 0,Y 368.991,Z 152.516,A -85,B 0,C 180,E1 -12797.742,E2 -12797.742} C_VEL
LIN {X 0,Y 368.91,Z 152.529,A -85,B 0,C 180,E1 -12801.22,E2 -12801.22} C_VEL
LIN {X 0,Y 368.954,Z 152.526,A -85,B 0,C 180,E1 -12804.775,E2 -12804.775} C_VEL
LIN {X 0,Y 368.962,Z 152.525,A -85,B 0,C 180,E1 -12807.203,E2 -12807.203} C_VEL
LIN {X 0,Y 368.918,Z 152.531,A -85,B 0,C 180,E1 -12809.689,E2 -12809.689} C_VEL
LIN {X 0,Y 368.896,Z 152.533,A -85,B 0,C 180,E1 -12813.043,E2 -12813.043} C_VEL
LIN {X 0,Y 368.916,Z 152.535,A -85,B 0,C 180,E1 -12816.196,E2 -12816.196} C_VEL
LIN {X 0,Y 368.901,Z 152.531,A -85,B 0,C 180,E1 -12818.953,E2 -12818.953} C_VEL
LIN {X 0,Y 368.879,Z 152.538,A -85,B 0,C 180,E1 -12822.009,E2 -12822.009} C_VEL
LIN {X 0,Y 368.913,Z 152.586,A -85,B 0,C 180,E1 -12824.41,E2 -12824.41} C_VEL
LIN {X 0,Y 371.327,Z 163.244,A -85,B 0,C 180,E1 -12827.464,E2 -12827.464} C_VEL
LIN {X 0,Y 376.121,Z 175.16,A -85,B 0,C 180,E1 -12828.094,E2 -12828.094} C_VEL
LIN {X 0,Y 379.15,Z 189.065,A -85,B 0,C 180,E1 -12828.611,E2 -12828.611} C_VEL
LIN {X 0,Y 377.407,Z 271.17,A -85,B 0,C 180,E1 -12830.245,E2 -12830.245} C_VEL
LIN {X 0,Y 376.809,Z 284.385,A -85,B 0,C 180,E1 -12830.73,E2 -12830.73} C_VEL
LIN {X 0,Y 376.05,Z 297.13,A -85,B 0,C 180,E1 -12831.427,E2 -12831.427} C_VEL
LIN {X 0,Y 375.042,Z 309.008,A -85,B 0,C 180,E1 -12832.311,E2 -12832.311} C_VEL
LIN {X 0,Y 373.937,Z 319.816,A -85,B 0,C 180,E1 -12833.34,E2 -12833.34} C_VEL
LIN {X 0,Y 372.779,Z 330.157,A -85,B 0,C 180,E1 -12834.568,E2 -12834.568} C_VEL
LIN {X 0,Y 371.6,Z 339.739,A -85,B 0,C 180,E1 -12835.992,E2 -12835.992} C_VEL
LIN {X 0,Y 370.499,Z 348.415,A -85,B 0,C 180,E1 -12837.597,E2 -12837.597} C_VEL
LIN {X 0,Y 369.482,Z 356.229,A -85,B 0,C 180,E1 -12839.415,E2 -12839.415} C_VEL
LIN {X 0,Y 368.712,Z 362.345,A -85,B 0,C 180,E1 -12841.258,E2 -12841.258} C_VEL
LIN {X 0,Y 368.076,Z 367.542,A -85,B 0,C 180,E1 -12843.34,E2 -12843.34} C_VEL
LIN {X 0,Y 367.686,Z 370.666,A -85,B 0,C 180,E1 -12845.133,E2 -12845.133} C_VEL
LIN {X 0,Y 367.493,Z 372.398,A -85,B 0,C 180,E1 -12846.628,E2 -12846.628} C_VEL
LIN {X 0,Y 367.317,Z 373.589,A -85,B 0,C 180,E1 -12848.683,E2 -12848.683} C_VEL
LIN {X 0,Y 367.306,Z 373.626,A -85,B 0,C 180,E1 -12849.854,E2 -12849.854} C_VEL
LIN {X 0,Y 367.265,Z 373.246,A -85,B 0,C 180,E1 -12851.016,E2 -12851.016} C_VEL
LIN {X 0,Y 367.407,Z 371.534,A -85,B 0,C 180,E1 -12853.022,E2 -12853.022} C_VEL
LIN {X 0,Y 367.668,Z 368.365,A -85,B 0,C 180,E1 -12855.045,E2 -12855.045} C_VEL
LIN {X 0,Y 367.985,Z 364.114,A -85,B 0,C 180,E1 -12856.91,E2 -12856.91} C_VEL
LIN {X 0,Y 368.327,Z 359.532,A -85,B 0,C 180,E1 -12858.443,E2 -12858.443} C_VEL
LIN {X 0,Y 368.81,Z 353.232,A -85,B 0,C 180,E1 -12860.125,E2 -12860.125} C_VEL
LIN {X 0,Y 369.507,Z 345.435,A -85,B 0,C 180,E1 -12861.783,E2 -12861.783} C_VEL
LIN {X 0,Y 370.305,Z 337.245,A -85,B 0,C 180,E1 -12863.188,E2 -12863.188} C_VEL
LIN {X 0,Y 371.153,Z 327.379,A -85,B 0,C 180,E1 -12864.567,E2 -12864.567} C_VEL
LIN {X 0,Y 372.111,Z 316.347,A -85,B 0,C 180,E1 -12865.803,E2 -12865.803} C_VEL
LIN {X 0,Y 372.988,Z 303.985,A -85,B 0,C 180,E1 -12866.878,E2 -12866.878} C_VEL
LIN {X 0,Y 373.574,Z 292.152,A -85,B 0,C 180,E1 -12867.67,E2 -12867.67} C_VEL
LIN {X 0,Y 374.12,Z 279.356,A -85,B 0,C 180,E1 -12868.285,E2 -12868.285} C_VEL
LIN {X 0,Y 374.536,Z 265.945,A -85,B 0,C 180,E1 -12868.69,E2 -12868.69} C_VEL
LIN {X 0,Y 375.797,Z 186.236,A -85,B 0,C 180,E1 -12870.235,E2 -12870.235} C_VEL
LIN {X 0,Y 371.491,Z 164.552,A -85,B 0,C 180,E1 -12870.882,E2 -12870.882} C_VEL
LIN {X 0,Y 370.915,Z 162.63,A -85,B 0,C 180,E1 -12870.964,E2 -12870.964} C_VEL
LIN {X 0,Y 370.402,Z 159.211,A -85,B 0,C 180,E1 -12871.852,E2 -12871.852} C_VEL
LIN {X 0,Y 369.406,Z 157.339,A -85,B 0,C 180,E1 -12872.382,E2 -12872.382} C_VEL
LIN {X 0,Y 365.958,Z 154.947,A -85,B 0,C 180,E1 -12873.232,E2 -12873.232} C_VEL
LIN {X 0,Y 363.195,Z 153.826,A -85,B 0,C 180,E1 -12873.953,E2 -12873.953} C_VEL
LIN {X 0,Y 362.022,Z 153.429,A -85,B 0,C 180,E1 -12874.554,E2 -12874.554} C_VEL
LIN {X 0,Y 361.945,Z 153.396,A -85,B 0,C 180,E1 -12874.765,E2 -12874.765} C_VEL
LIN {X 0,Y 362.115,Z 153.375,A -85,B 0,C 180,E1 -12876.687,E2 -12876.687} C_VEL
LIN {X 0,Y 361.989,Z 153.394,A -85,B 0,C 180,E1 -12880.063,E2 -12880.063} C_VEL
LIN {X 0,Y 361.946,Z 153.401,A -85,B 0,C 180,E1 -12883.868,E2 -12883.868} C_VEL
LIN {X 0,Y 361.891,Z 153.406,A -85,B 0,C 180,E1 -12887.903,E2 -12887.903} C_VEL
LIN {X 0,Y 361.842,Z 153.414,A -85,B 0,C 180,E1 -12891.656,E2 -12891.656} C_VEL
LIN {X 0,Y 361.847,Z 153.413,A -85,B 0,C 180,E1 -12895.297,E2 -12895.297} C_VEL
LIN {X 0,Y 361.852,Z 153.411,A -85,B 0,C 180,E1 -12899.074,E2 -12899.074} C_VEL
LIN {X 0,Y 361.844,Z 153.412,A -85,B 0,C 180,E1 -12902.946,E2 -12902.946} C_VEL
LIN {X 0,Y 361.86,Z 153.409,A -85,B 0,C 180,E1 -12905.638,E2 -12905.638} C_VEL
LIN {X 0,Y 361.823,Z 153.417,A -85,B 0,C 180,E1 -12909.018,E2 -12909.018} C_VEL
LIN {X 0,Y 361.827,Z 153.415,A -85,B 0,C 180,E1 -12912.831,E2 -12912.831} C_VEL
LIN {X 0,Y 361.812,Z 153.413,A -85,B 0,C 180,E1 -12915.948,E2 -12915.948} C_VEL
LIN {X 0,Y 361.809,Z 153.415,A -85,B 0,C 180,E1 -12919.25,E2 -12919.25} C_VEL
